// TwinCAT 3 PLC project PLC
// ProgramVersion: 3.1.4023.0
// libraries:
//   Tc2_Standard, * (Beckhoff Automation GmbH)
//   Tc2_System, * (Beckhoff Automation GmbH)
//   Tc3_Module, * (Beckhoff Automation GmbH)
// project tree:
//   / PlcTask.TcTTO
//   POUs/ MAIN.TcPOU
//   DUTs/IO/PdoEntries/ Status_56B69FDC.TcDUT (not stored), Inputs_62625F94.TcDUT (not stored), Ctrl_F19EAB21.TcDUT (not stored), Inputs_102D1D08.TcDUT (not stored), Status_642C2ED1.TcDUT (not stored), Ctrl_B05F80DF.TcDUT (not stored), Outputs_A910484D.TcDUT (not stored), Ctrl_77460BD3.TcDUT (not stored), Channel_EA8D33D7.TcDUT (not stored), Channel_D623F56C.TcDUT (not stored), Status_D9DC9C1B.TcDUT (not stored), Control_4E83000D.TcDUT (not stored), Status_8D3FCD23.TcDUT (not stored), Control_87176C1F.TcDUT (not stored), Device_status_8568DBCA.TcDUT (not stored), Outputs_Group_78994C08.TcDUT (not stored), Outputs_Channel_78994C08.TcDUT (not stored), Status_F2CE6D91.TcDUT (not stored), STATUS_B0753356.TcDUT (not stored), Status_237FCB0F.TcDUT (not stored), Setting_24C04940.TcDUT (not stored), Ctrl_56BB2DF2.TcDUT (not stored), Status_51F0A924.TcDUT (not stored), Settings_24C04940.TcDUT (not stored), Control_18D542D9.TcDUT (not stored), Status_439F40C3.TcDUT (not stored), Status_B0753356.TcDUT (not stored), Status_68C33E99.TcDUT (not stored), Status_7BCDA921.TcDUT (not stored), Ctrl_B9DDD3FF.TcDUT (not stored), Status_ACC8459F.TcDUT (not stored), Status_536663CA.TcDUT (not stored), Status_C03E2495.TcDUT (not stored), Status_A9D94975.TcDUT (not stored), Control_D500AB79.TcDUT (not stored), Status_81FEA767.TcDUT (not stored), Status_36731094.TcDUT (not stored), Status_6D6CFE20.TcDUT (not stored), Control_6EF2C5D0.TcDUT (not stored), Status_D8D782C3.TcDUT (not stored), Status_E2E79E85.TcDUT (not stored), Status_2E3946CF.TcDUT (not stored), Counter_value_E1FCE22B.TcDUT (not stored), Control_BD9A418F.TcDUT (not stored), Status_396FCBA0.TcDUT (not stored), Status_AA25F79C.TcDUT (not stored), Control_D4F3D880.TcDUT (not stored), Status_770B5231.TcDUT (not stored), Control_A35B59FC.TcDUT (not stored), Status_3E6F3FF3.TcDUT (not stored), Status_3BE3BF26.TcDUT (not stored), Control_135F4E52.TcDUT (not stored), Status_56494C1D.TcDUT (not stored), Status_3D84275F.TcDUT (not stored), Ctrl_71604E86.TcDUT (not stored), Ctrl_1EFB4D3B.TcDUT (not stored), Status_E3E7FD12.TcDUT (not stored), Slave_1_Inputs_2C3058A8.TcDUT (not stored), Slave_2_Inputs_413F454C.TcDUT (not stored), Slave_3_Inputs_9985457D.TcDUT (not stored), Slave_4_Inputs_9B217E84.TcDUT (not stored), Slave_5_Inputs_439B7EB5.TcDUT (not stored), Slave_6_Inputs_2E946351.TcDUT (not stored), Slave_7_Inputs_F62E6360.TcDUT (not stored), Slave_8_Inputs_2BDC14A3.TcDUT (not stored), Slave_9_Inputs_F3661492.TcDUT (not stored), Slave_10_Inputs_01E65E7D.TcDUT (not stored), Slave_11_Inputs_D274DB97.TcDUT (not stored), Slave_12_Inputs_A202481E.TcDUT (not stored), Slave_13_Inputs_7190CDF4.TcDUT (not stored), Slave_14_Inputs_42EF6F0C.TcDUT (not stored), Slave_15_Inputs_917DEAE6.TcDUT (not stored), Slave_16_Inputs_E10B796F.TcDUT (not stored), Slave_17_Inputs_3299FC85.TcDUT (not stored), Slave_18_Inputs_87F43C9F.TcDUT (not stored), Slave_19_Inputs_5466B975.TcDUT (not stored), Slave_20_Inputs_97C1CA9A.TcDUT (not stored), Slave_21_Inputs_44534F70.TcDUT (not stored), Slave_22_Inputs_3425DCF9.TcDUT (not stored), Slave_23_Inputs_E7B75913.TcDUT (not stored), Slave_24_Inputs_D4C8FBEB.TcDUT (not stored), Slave_25_Inputs_075A7E01.TcDUT (not stored), Slave_26_Inputs_772CED88.TcDUT (not stored), Slave_27_Inputs_A4BE6862.TcDUT (not stored), Slave_28_Inputs_11D3A878.TcDUT (not stored), Slave_29_Inputs_C2412D92.TcDUT (not stored), Slave_30_Inputs_199C4DAA.TcDUT (not stored), Slave_31_Inputs_CA0EC840.TcDUT (not stored), Slave_1_Outputs_820A30FD.TcDUT (not stored), Slave_2_Outputs_EF052D19.TcDUT (not stored), Slave_3_Outputs_37BF2D28.TcDUT (not stored), Slave_4_Outputs_351B16D1.TcDUT (not stored), Slave_5_Outputs_EDA116E0.TcDUT (not stored), Slave_6_Outputs_80AE0B04.TcDUT (not stored), Slave_7_Outputs_58140B35.TcDUT (not stored), Slave_8_Outputs_85E67CF6.TcDUT (not stored), Slave_9_Outputs_5D5C7CC7.TcDUT (not stored), Slave_10_Outputs_0FEEBBCA.TcDUT (not stored), Slave_11_Outputs_DC7C3E20.TcDUT (not stored), Slave_12_Outputs_AC0AADA9.TcDUT (not stored), Slave_13_Outputs_7F982843.TcDUT (not stored), Slave_14_Outputs_4CE78ABB.TcDUT (not stored), Slave_15_Outputs_9F750F51.TcDUT (not stored), Slave_16_Outputs_EF039CD8.TcDUT (not stored), Slave_17_Outputs_3C911932.TcDUT (not stored), Slave_18_Outputs_89FCD928.TcDUT (not stored), Slave_19_Outputs_5A6E5CC2.TcDUT (not stored), Slave_20_Outputs_99C92F2D.TcDUT (not stored), Slave_21_Outputs_4A5BAAC7.TcDUT (not stored), Slave_22_Outputs_3A2D394E.TcDUT (not stored), Slave_23_Outputs_E9BFBCA4.TcDUT (not stored), Slave_24_Outputs_DAC01E5C.TcDUT (not stored), Slave_25_Outputs_09529BB6.TcDUT (not stored), Slave_26_Outputs_7924083F.TcDUT (not stored), Slave_27_Outputs_AAB68DD5.TcDUT (not stored), Slave_28_Outputs_1FDB4DCF.TcDUT (not stored), Slave_29_Outputs_CC49C825.TcDUT (not stored), Slave_30_Outputs_1794A81D.TcDUT (not stored), Slave_31_Outputs_C4062DF7.TcDUT (not stored), Status_182674C6.TcDUT (not stored), Status_B6795845.TcDUT (not stored), Control_F189B737.TcDUT (not stored), Control_C948E0F2.TcDUT (not stored), Status_8CBE219F.TcDUT (not stored), Status_1E008DB9.TcDUT (not stored), Control_5FD4673D.TcDUT (not stored), Status_36C8BFF1.TcDUT (not stored), Status_FCAFFB9E.TcDUT (not stored), Control_534FEB19.TcDUT (not stored), Status_1D9409A4.TcDUT (not stored), Status_26C2D68E.TcDUT (not stored), Control_854091F6.TcDUT (not stored), Status_8AD1B54B.TcDUT (not stored), Control_0B2F8B70.TcDUT (not stored), FSOE_8C3E79C6.TcDUT (not stored), FSOE_3054F843.TcDUT (not stored), Status_8A0522A0.TcDUT (not stored), Ctrl_8F963B2D.TcDUT (not stored), Status_FCC1AD92.TcDUT (not stored), Status_6F0FEDB3.TcDUT (not stored), Control_DAEE1D52.TcDUT (not stored), Status_5E172F14.TcDUT (not stored), Status_CDD96F35.TcDUT (not stored), Status_B8381171.TcDUT (not stored), Status_7097155E.TcDUT (not stored), Control_7786EF9F.TcDUT (not stored), Status_70E023F8.TcDUT (not stored), Control_A8DDCD82.TcDUT (not stored), Status_EBCAF3EC.TcDUT (not stored), Control_254441A5.TcDUT (not stored), Status_72C27E80.TcDUT (not stored), Status_6BD97C37.TcDUT (not stored), Status_3BF44A81.TcDUT (not stored), Control_7648F432.TcDUT (not stored), Status_9AF2E088.TcDUT (not stored), Control_12F99C76.TcDUT (not stored), FSOE_BDDA3532.TcDUT (not stored), FSOE_EE2DB9C3.TcDUT (not stored), FSOE_046F804E.TcDUT (not stored), FSOE_F7635245.TcDUT (not stored), Status_05CE4FB5.TcDUT (not stored), Ctrl_AEDC374E.TcDUT (not stored), STATUS_1538B4EA.TcDUT (not stored), STATUS_522E84CD.TcDUT (not stored), STATUS_58431BA9.TcDUT (not stored), Status_543010BE.TcDUT (not stored), Samples_F24E104A.TcDUT (not stored), StartTimeNextLatch_02E0C1C8.TcDUT (not stored), U1_STATUS_B0753356.TcDUT (not stored), U1_SAMPLES_2D13B74B.TcDUT (not stored), I1_STATUS_B0753356.TcDUT (not stored), I1_SAMPLES_2D13B74B.TcDUT (not stored), U2_STATUS_B0753356.TcDUT (not stored), U2_SAMPLES_2D13B74B.TcDUT (not stored), I2_STATUS_B0753356.TcDUT (not stored), I2_SAMPLES_2D13B74B.TcDUT (not stored), U3_STATUS_B0753356.TcDUT (not stored), U3_SAMPLES_2D13B74B.TcDUT (not stored), I3_STATUS_B0753356.TcDUT (not stored), I3_SAMPLES_2D13B74B.TcDUT (not stored), U1_Status_DC903920.TcDUT (not stored), U1_Samples_2D13B74B.TcDUT (not stored), I1_Status_DC903920.TcDUT (not stored), I1_Samples_2D13B74B.TcDUT (not stored), U2_Status_DC903920.TcDUT (not stored), U2_Samples_2D13B74B.TcDUT (not stored), I2_Status_DC903920.TcDUT (not stored), I2_Samples_2D13B74B.TcDUT (not stored), U3_Status_DC903920.TcDUT (not stored), U3_Samples_2D13B74B.TcDUT (not stored), I3_Status_DC903920.TcDUT (not stored), I3_Samples_2D13B74B.TcDUT (not stored), U1_Samples_25492287.TcDUT (not stored), I1_Samples_25492287.TcDUT (not stored), U2_Samples_25492287.TcDUT (not stored), I2_Samples_25492287.TcDUT (not stored), U3_Samples_25492287.TcDUT (not stored), I3_Samples_25492287.TcDUT (not stored), U1_Samples_1109DCAA.TcDUT (not stored), I1_Samples_1109DCAA.TcDUT (not stored), U2_Samples_1109DCAA.TcDUT (not stored), I2_Samples_1109DCAA.TcDUT (not stored), U3_Samples_1109DCAA.TcDUT (not stored), I3_Samples_1109DCAA.TcDUT (not stored), High_Current_Range_48967762.TcDUT (not stored), Status_7BCA2D07.TcDUT (not stored), Ctrl_E6581599.TcDUT (not stored), Status_3035BE2E.TcDUT (not stored), Control_4AE59EC2.TcDUT (not stored)
//   DUTs/IO/PDOs/ InfoData_6F19DB2B.TcDUT (not stored), Channel_830843C1.TcDUT (not stored), WcState_9091E0EB.TcDUT (not stored), Channel_31CEFA7F.TcDUT (not stored), EMPTY_STRUCTURE.TcDUT (not stored), DC_1A6E6625.TcDUT (not stored), InfoData_A7436BC6.TcDUT (not stored), Latch_8E413295.TcDUT (not stored), Latch_39BD7C7C.TcDUT (not stored), Latch_0465F916.TcDUT (not stored), Ch1_CycleCount_9DBE2BC5.TcDUT (not stored), Ch1_Input_FFC4CE24.TcDUT (not stored), Ch2_CycleCount_976A51B5.TcDUT (not stored), Ch2_Input_78ADA90C.TcDUT (not stored), NextSync1Time_EE185E17.TcDUT (not stored), MTI_Inputs_10x_Channel_C3ED30FD.TcDUT (not stored), MTI_Outputs_Channel_0F1028A1.TcDUT (not stored), InfoData_BEF6B88E.TcDUT (not stored), MTI_Inputs_1x_Channel_CC1B212F.TcDUT (not stored), MTO_Inputs_Channel_53C09E8B.TcDUT (not stored), MTO_Outputs_10x_Channel_232E0117.TcDUT (not stored), MTO_Outputs_10x_Channel_A3C0C022.TcDUT (not stored), Channel_42CA91F7.TcDUT (not stored), WcState_0B2B16F9.TcDUT (not stored), DIG_Diag_Inputs_58F3E2A8.TcDUT (not stored), DIG_Inputs_Device_A1F150A9.TcDUT (not stored), DIG_Outputs_F9744C66.TcDUT (not stored), InfoData_32EB74EA.TcDUT (not stored), Diag_A72B1E17.TcDUT (not stored), Channel_54BE63B3.TcDUT (not stored), DOX_Status_Channel_09DD45C8.TcDUT (not stored), DOX_Control_Channel_A74F2363.TcDUT (not stored), DOX_Status_Channel_6FDDBA98.TcDUT (not stored), DOX_Control_Channel_E6930641.TcDUT (not stored), DC_Sync_Activate_FA2D2910.TcDUT (not stored), DC_Sync_Start_9CCB0E51.TcDUT (not stored), DC_Sync_Start_E82E9233.TcDUT (not stored), Cycle_Counter_2C233804.TcDUT (not stored), Sample_3C4603C7.TcDUT (not stored), CycCount0_2C233804.TcDUT (not stored), Sample_0023574C.TcDUT (not stored), CycCount1_2C233804.TcDUT (not stored), Sample_07D5B44A.TcDUT (not stored), CycCount0_AF431CE0.TcDUT (not stored), CycCount1_A8B5FFE6.TcDUT (not stored), StartTimeNextOutput_228767F4.TcDUT (not stored), Inputs_298FB92D.TcDUT (not stored), DO_Inputs_Device_4A9049C5.TcDUT (not stored), DO_Group_1_Outputs_59D8C01C.TcDUT (not stored), DO_Group_2_Outputs_82808288.TcDUT (not stored), DIG_Diag_Inputs_F289D615.TcDUT (not stored), DIG_Outputs_B9300CB6.TcDUT (not stored), Diagnostic_A72B1E17.TcDUT (not stored), DO_Group_1_Outputs_07009A9C.TcDUT (not stored), DO_Group_2_Outputs_3033EF65.TcDUT (not stored), DO_Group_3_Outputs_22DD3C32.TcDUT (not stored), DO_Group_4_Outputs_5E550497.TcDUT (not stored), AI_Inputs_Channel_10B8F80A.TcDUT (not stored), AI_Inputs_Channel_45213104.TcDUT (not stored), AI_Inputs_45213104.TcDUT (not stored), Ch1_Status_75824485.TcDUT (not stored), Ch1_Sample_A71DD501.TcDUT (not stored), Ch2_Status_75824485.TcDUT (not stored), Ch2_Sample_9F6886E6.TcDUT (not stored), Next_Sync1_Time_434371C2.TcDUT (not stored), Sample_Count_C25D5F38.TcDUT (not stored), NextSync1Time_9AFDC275.TcDUT (not stored), Sample_Count_EA88CAD9.TcDUT (not stored), SAI_Inputs_3A838E11.TcDUT (not stored), SAI_Range_C3200E78.TcDUT (not stored), SAI_Range_3710D747.TcDUT (not stored), SAI_Inputs_84B29FE9.TcDUT (not stored), SAI_Range_BDBF6DA9.TcDUT (not stored), SAI_Range_2A187FC5.TcDUT (not stored), SAI_Feedback_BDBF6DA9.TcDUT (not stored), SAI_Inputs_Channel_9DCD6557.TcDUT (not stored), SAI_Range_Channel_BDBF6DA9.TcDUT (not stored), SAI_Inputs_Real_Channel_CCECF13D.TcDUT (not stored), AI_Standard_Channel_A8DF64E3.TcDUT (not stored), TC_Inputs_Channel_204FE750.TcDUT (not stored), AI_Standard_Channel_4A394481.TcDUT (not stored), RMB_Status_C0E100AA.TcDUT (not stored), RMB_Value_INT_E9189C4B.TcDUT (not stored), RMB_Control_CC49845C.TcDUT (not stored), AO_Output_Channel_BA7EBB7C.TcDUT (not stored), Channel_5F9B7EA6.TcDUT (not stored), Channel_4E63E14D.TcDUT (not stored), Channel_DD2C734A.TcDUT (not stored), SSI_Inputs_0E3D8E33.TcDUT (not stored), SSI_Inputs_3B70A311.TcDUT (not stored), SSI_Inputs_8BC18DAC.TcDUT (not stored), SSI_Inputs_Channel_0E3D8E33.TcDUT (not stored), SSI_Inputs_Channel_EDA16284.TcDUT (not stored), ENC_Status_1E2673DC.TcDUT (not stored), ENC_Control_64DD586E.TcDUT (not stored), FB_Inputs_Channel_74050988.TcDUT (not stored), IND_Inputs_Channel_BBE8401F.TcDUT (not stored), IND_Outputs_Channel_02FDE6C9.TcDUT (not stored), Channel_B90637B9.TcDUT (not stored), Channel_C6781B15.TcDUT (not stored), Inputs_B90637B9.TcDUT (not stored), Outputs_C6781B15.TcDUT (not stored), ENC_Status_compact_D1AA7539.TcDUT (not stored), ENC_Control_compact_6FDDC669.TcDUT (not stored), ENC_Status_compact_6F424558.TcDUT (not stored), ENC_Control_compact_21E2D14D.TcDUT (not stored), ENC_Status_compact_7D3464F3.TcDUT (not stored), ENC_Status_compact_4198EF3B.TcDUT (not stored), ENC_Status_4E2088B9.TcDUT (not stored), ENC_NextSync1Time_9AFDC275.TcDUT (not stored), ENC_TxPdo_1_Samples_Counter_value_215818C6.TcDUT (not stored), ENC_Control_14E3EF4F.TcDUT (not stored), ENC_Inputs_3399C5AA.TcDUT (not stored), ENC_Inputs_24B63C53.TcDUT (not stored), ENC_Outputs_2E45048F.TcDUT (not stored), ENC_Status_Channel_10A67E52.TcDUT (not stored), ENC_Control_Channel_4C8A7395.TcDUT (not stored), ENC_Status_Channel_04F16FC0.TcDUT (not stored), ENC_Control_Channel_B930862D.TcDUT (not stored), ENC_Inputs_561E041F.TcDUT (not stored), ENC_Inputs_B3536485.TcDUT (not stored), ENC_Outputs_21E2D14D.TcDUT (not stored), ENC_Status_AC51C0C0.TcDUT (not stored), ENC_Filtered_latch_2CF1EFF6.TcDUT (not stored), ENC_Control_EB665241.TcDUT (not stored), ENC_Inputs_F139456B.TcDUT (not stored), ENC_Outputs_6FDDC669.TcDUT (not stored), ENC_Status_compact_B3536485.TcDUT (not stored), ENC_Status_compact_Channel_0EF60376.TcDUT (not stored), ENC_Period_Channel_24B63C53.TcDUT (not stored), ENC_Control_compact_Channel_245CB94B.TcDUT (not stored), ENC_Status_compact_Channel_FA024B16.TcDUT (not stored), ENC_Control_compact_Channel_2ED727EF.TcDUT (not stored), Inputs_6C2FC202.TcDUT (not stored), Outputs_5D00B5E7.TcDUT (not stored), COM_Inputs_3801C95E.TcDUT (not stored), COM_Outputs_DEF408EC.TcDUT (not stored), COM_Inputs_Channel_3801C95E.TcDUT (not stored), COM_Outputs_Channel_EADA2E0D.TcDUT (not stored), COM_TxPDO_Map_Inputs_Channel_3801C95E.TcDUT (not stored), COM_RxPDO_Map_Outputs_Channel_EADA2E0D.TcDUT (not stored), COM_TxPDO_Map_Inputs_3801C95E.TcDUT (not stored), COM_RxPDO_Map_Outputs_DEF408EC.TcDUT (not stored), Status_EF5E6C28.TcDUT (not stored), Control_88301954.TcDUT (not stored), Status_07D3AAF6.TcDUT (not stored), Control_DAFD38E0.TcDUT (not stored), DIS_Inputs_E0E384E3.TcDUT (not stored), DIS_Outputs_6C9BFFEE.TcDUT (not stored), ASI_Inputs_Device_7F2828A5.TcDUT (not stored), ASI_Status_8C8FBBB4.TcDUT (not stored), ASI_Outputs_Device_16036E19.TcDUT (not stored), ASI_Control_F45BBE2B.TcDUT (not stored), ASI_Status_279C3903.TcDUT (not stored), ASI_Control_2BED1893.TcDUT (not stored), DeviceState_Inputs_4751FF76.TcDUT (not stored), InfoData_90184F0C.TcDUT (not stored), DeviceState_Inputs_Device_A1210598.TcDUT (not stored), Module_1_DeviceState_Inputs_Device_5322301C.TcDUT (not stored), Module_2_DeviceState_Inputs_BD6C7035.TcDUT (not stored), ENC_Status_compact_3C6E2C44.TcDUT (not stored), STM_Status_36ED096F.TcDUT (not stored), ENC_Control_compact_2E82BC43.TcDUT (not stored), STM_Control_5A8B5016.TcDUT (not stored), STM_Velocity_A47A3F41.TcDUT (not stored), InfoData_8DF4E0C5.TcDUT (not stored), InfoData_6538CF5F.TcDUT (not stored), AI_Standard_Channel_205D8A06.TcDUT (not stored), InfoData_939F71B6.TcDUT (not stored), ENC_Status_compact_4D066E1A.TcDUT (not stored), STM_Status_DE0D6B37.TcDUT (not stored), STM_Control_BA4CE352.TcDUT (not stored), STM_Status_5B5B2475.TcDUT (not stored), FB_Position_3FA094ED.TcDUT (not stored), DRV_Statusword_9B36FDFC.TcDUT (not stored), DRV_Following_error_actual_value_5AA320BF.TcDUT (not stored), DRV_Controlword_F3F14721.TcDUT (not stored), DRV_Target_position_05240F14.TcDUT (not stored), InfoData_6185D47C.TcDUT (not stored), PowerOK_830843C1.TcDUT (not stored), PowerOK_CEB2FD12.TcDUT (not stored), FuseError_1EC650DA.TcDUT (not stored), OCP_Inputs_8CCE65FB.TcDUT (not stored), OCP_Outputs_01014934.TcDUT (not stored), OCP_Inputs_Channel_8CCE65FB.TcDUT (not stored), OCP_Outputs_Channel_01014934.TcDUT (not stored), OCP_Inputs_Channel_794A321B.TcDUT (not stored), Status_Us_B1E819A2.TcDUT (not stored), Status_Up_B1E819A2.TcDUT (not stored), Status_Uo_B8D9F2FA.TcDUT (not stored), Status_Up_DB353128.TcDUT (not stored), Status_Us_DB353128.TcDUT (not stored), Status_Us_449D6AB5.TcDUT (not stored), Status_Uo_449D6AB5.TcDUT (not stored), BCT_Inputs_28C1780C.TcDUT (not stored), BCT_Inputs_8E55234D.TcDUT (not stored), BCT_Inputs_4B987895.TcDUT (not stored), BCT_Inputs_8B1D510C.TcDUT (not stored), BCT_Inputs_7ACE8FA6.TcDUT (not stored), CNT_Inputs_7D4495CD.TcDUT (not stored), CNT_Outputs_EB14A675.TcDUT (not stored), CNT_Inputs_147BF88E.TcDUT (not stored), CNT_Inputs_B6C38E71.TcDUT (not stored), CNT_Outputs_458039AE.TcDUT (not stored), CNT_Inputs_Channel_21E1BB39.TcDUT (not stored), CNT_Outputs_Channel_774A30BC.TcDUT (not stored), CNT_Inputs_Channel_54FF2F1E.TcDUT (not stored), CNT_Outputs_Channel_550BB6DF.TcDUT (not stored), FSoE_Inputs_8E27404E.TcDUT (not stored), FSoE_Outputs_5936ECC6.TcDUT (not stored), FSLOGIC_Inputs_EEE9388E.TcDUT (not stored), Module_1_FSOE_79A9B6A8.TcDUT (not stored), Module_2_FSLOGIC_DEAB4522.TcDUT (not stored), PWM_Outputs_Channel_4C6289CD.TcDUT (not stored), PWM_Inputs_Channel_4239F652.TcDUT (not stored), PWM_SysTime_Channel_10DC6945.TcDUT (not stored), PWM_Per_DC_Outputs_Channel_C8E719F3.TcDUT (not stored), Inputs_A3335424.TcDUT (not stored), Outputs_8F8B60FA.TcDUT (not stored), PTO_Status_B6D696E0.TcDUT (not stored), ENC_Status_compact_EA7A730E.TcDUT (not stored), PTO_Control_392B4D2E.TcDUT (not stored), PTO_Target_compact_5C359F7D.TcDUT (not stored), ENC_Control_compact_245CB94B.TcDUT (not stored), PTO_Status_B24E260C.TcDUT (not stored), ENC_Status_compact_4C428F88.TcDUT (not stored), PTO_Control_9287F8E4.TcDUT (not stored), ENC_Control_compact_2ED727EF.TcDUT (not stored), PTO_Status_40B3051C.TcDUT (not stored), ENC_Status_compact_036460C9.TcDUT (not stored), PTO_Status_C6D3EC31.TcDUT (not stored), ENC_Status_compact_64F890EB.TcDUT (not stored), PLS_Status_A60F4933.TcDUT (not stored), ENC_Control_compact_DC4E290B.TcDUT (not stored), PLS_Control_compact_DC91A7B8.TcDUT (not stored), PTO_Status_E0EB10E8.TcDUT (not stored), PLS_Status_70E7A1E2.TcDUT (not stored), PLS_Control_compact_CD6E44DE.TcDUT (not stored), Inputs_0292EF13.TcDUT (not stored), Outputs_905E7D86.TcDUT (not stored), PTO_Status_Channel_E0EB10E8.TcDUT (not stored), ENC_Status_Channel_A9252C48.TcDUT (not stored), PTO_Control_Channel_9287F8E4.TcDUT (not stored), PTO_Target_Channel_1F6D5BC6.TcDUT (not stored), ENC_Control_Channel_686BB9DC.TcDUT (not stored), PWM_Status_Channel_2D1AF340.TcDUT (not stored), PWM_Control_Channel_63F162E4.TcDUT (not stored), PWM_Status_Channel_77939B11.TcDUT (not stored), PWM_Inputs_Channel_304DC245.TcDUT (not stored), PWM_Outputs_Channel_D6F04FBD.TcDUT (not stored), DOX_Status_AED8A12A.TcDUT (not stored), DOX_Control_75D5C9E2.TcDUT (not stored), DOX_Status_F52B34D3.TcDUT (not stored), DOX_Control_B191BB93.TcDUT (not stored), FSoE_Inputs_C161D7C0.TcDUT (not stored), FSoE_Outputs_F73BE43A.TcDUT (not stored), Outputs_A2CAA446.TcDUT (not stored), FIELDVOLTAGE_Field_Voltage_Status_9DC7C349.TcDUT (not stored), WcState_B516A264.TcDUT (not stored), Module_1_FSOE_7E34DB40.TcDUT (not stored), Module_2_FSOUT_1E8D1637.TcDUT (not stored), Module_3_DEVICEIO_5FA6B4E7.TcDUT (not stored), Module_4_FSLOGIC_DEAB4522.TcDUT (not stored), FSoE_Inputs_939ABF3D.TcDUT (not stored), FSoE_Outputs_3899B185.TcDUT (not stored), Outputs_8B1C946D.TcDUT (not stored), Module_1_FSOE_263516AE.TcDUT (not stored), Module_2_FSOUT_6D5CB05D.TcDUT (not stored), AI_Standard_EA9DF21E.TcDUT (not stored), AI_Standard_Channel_EA9DF21E.TcDUT (not stored), AI_Standard_A8DF64E3.TcDUT (not stored), Channel_7539AA33.TcDUT (not stored), Ch_1_Al_Inputs_4794C083.TcDUT (not stored), Ch_2_Al_Inputs_4794C083.TcDUT (not stored), Ch_1_A1FAE759.TcDUT (not stored), Ch_2_D9CD36D2.TcDUT (not stored), RTD_Inputs_EA9DF21E.TcDUT (not stored), RTD_Inputs_Channel_EA9DF21E.TcDUT (not stored), RTD_Inputs_Channel_9575FEA1.TcDUT (not stored), RTD_Standard_Channel_A8DF64E3.TcDUT (not stored), AI_Compact_Channel_80E77D6A.TcDUT (not stored), TC_Inputs_EA9DF21E.TcDUT (not stored), TC_Inputs_Channel_EA9DF21E.TcDUT (not stored), TC_Inputs_Channel_45213104.TcDUT (not stored), TC_Channel_9575FEA1.TcDUT (not stored), AIBridge_Inputs_555AA1E8.TcDUT (not stored), AISupply_Inputs_555AA1E8.TcDUT (not stored), RMB_Control_4997AEF6.TcDUT (not stored), PM_Inputs_Channel_6909D406.TcDUT (not stored), PM_Status_data_0FD072A0.TcDUT (not stored), PM_Outputs_Channel_E5FBDE30.TcDUT (not stored), PM_Inputs_Channel_2468BF1D.TcDUT (not stored), PM_Inputs_Channel_2F868086.TcDUT (not stored), PM_Status_data_2A9514CB.TcDUT (not stored), PM_Inputs_Channel_345EAE54.TcDUT (not stored), PM_Inputs_Auxiliary_392D510B.TcDUT (not stored), PM_Outputs_Auxiliary_6BC1946F.TcDUT (not stored), PM_Inputs_Auxiliary_3661DB6D.TcDUT (not stored), Total_Status_1ACE98F0.TcDUT (not stored), Total_Advanced_3B87F467.TcDUT (not stored), Total_Active_C9A69AC1.TcDUT (not stored), Total_Apparent_8F93F985.TcDUT (not stored), Total_Reactive_EF01DEFD.TcDUT (not stored), Total_Statistic_Power_092925BE.TcDUT (not stored), Total_Statistic_PQF_E0243244.TcDUT (not stored), Total_Interval_Energy_37FCCEB0.TcDUT (not stored), Interval_1578BBD4.TcDUT (not stored), Total_Interval_1578BBD4.TcDUT (not stored), Total_Active_Reduced_0E616AE5.TcDUT (not stored), Total_Apparent_Reduced_4B7F3014.TcDUT (not stored), Total_Reactive_Reduced_207ED80C.TcDUT (not stored), Total_Interval_Energy_Reduced_B0A0CDD8.TcDUT (not stored), L1_Status_61BE8896.TcDUT (not stored), L1_Basic_665874DE.TcDUT (not stored), L1_Power_22301EDD.TcDUT (not stored), L1_Timing_CCFF711F.TcDUT (not stored), L2_Status_61BE8896.TcDUT (not stored), L2_Basic_665874DE.TcDUT (not stored), L2_Power_22301EDD.TcDUT (not stored), L2_Timing_CCFF711F.TcDUT (not stored), L3_Status_61BE8896.TcDUT (not stored), L3_Basic_665874DE.TcDUT (not stored), L3_Power_22301EDD.TcDUT (not stored), L3_Timing_CCFF711F.TcDUT (not stored), Total_Basic_FC2CFF17.TcDUT (not stored), Total_Active_F9B49EA1.TcDUT (not stored), Total_L_L_Voltage_28813519.TcDUT (not stored), Total_Total_L_L_Voltage_28813519.TcDUT (not stored), I1_Current_AFE1DFA2.TcDUT (not stored), I2_Current_AFE1DFA2.TcDUT (not stored), I3_Current_AFE1DFA2.TcDUT (not stored), I4_Current_AFE1DFA2.TcDUT (not stored), I5_Current_AFE1DFA2.TcDUT (not stored), I6_Current_AFE1DFA2.TcDUT (not stored), Total_Basic_F53F9C95.TcDUT (not stored), Total_Status_A62BD506.TcDUT (not stored), L1_Status_12B1E6BB.TcDUT (not stored), L2_Status_12B1E6BB.TcDUT (not stored), L3_Status_12B1E6BB.TcDUT (not stored), Total_Status_AD43C3B9.TcDUT (not stored), L1_Basic_9F3F6F48.TcDUT (not stored), L2_Basic_9F3F6F48.TcDUT (not stored), L3_Basic_9F3F6F48.TcDUT (not stored), PAI_Status_Channel_AE4AC104.TcDUT (not stored), PAI_Samples_EEA51725.TcDUT (not stored), PAI_Timestamp_6DC4D296.TcDUT (not stored), L1_Voltage_Status_784F03AD.TcDUT (not stored), L1_Voltage_Samples_ED678DEE.TcDUT (not stored), L1_Current_Samples_89E07818.TcDUT (not stored), L1_Current_Samples_3209B12F.TcDUT (not stored), L2_Voltage_Status_0626A010.TcDUT (not stored), L2_Voltage_Samples_D91109BE.TcDUT (not stored), L2_Current_Status_F789DBA5.TcDUT (not stored), L2_Current_Samples_067F357F.TcDUT (not stored), L3_Voltage_Status_2C01C17B.TcDUT (not stored), L3_Voltage_Samples_CAC3758E.TcDUT (not stored), L3_Current_Status_DDAEBACE.TcDUT (not stored), L3_Current_Samples_15AD494F.TcDUT (not stored), AI_Timestamp_NextSync1Time_9AFDC275.TcDUT (not stored), AI_CycleCount_B1A935A2.TcDUT (not stored), L1_Current_Status_89E07818.TcDUT (not stored), AI_Sample_Count_B1A935A2.TcDUT (not stored), L1_Voltage_Status_7371B043.TcDUT (not stored), L1_Voltage_Samples_926B408D.TcDUT (not stored), L1_Current_Status_82DECBF6.TcDUT (not stored), L1_Current_Samples_4D057C4C.TcDUT (not stored), L2_Voltage_Status_0D1813FE.TcDUT (not stored), L2_Voltage_Samples_A61DC4DD.TcDUT (not stored), L2_Current_Status_FCB7684B.TcDUT (not stored), L2_Current_Samples_7973F81C.TcDUT (not stored), L3_Voltage_Status_273F7295.TcDUT (not stored), L3_Voltage_Samples_B5CFB8ED.TcDUT (not stored), L3_Current_Status_D6900920.TcDUT (not stored), L3_Current_Samples_6AA1842C.TcDUT (not stored), AI_NextSync1Time_6DC4D296.TcDUT (not stored), AI_Sample_Count_EA88CAD9.TcDUT (not stored), L1_Voltage_Samples_41AEB7FF.TcDUT (not stored), L1_Current_Samples_9EC08B3E.TcDUT (not stored), L2_Voltage_Samples_75D833AF.TcDUT (not stored), L2_Current_Samples_AAB60F6E.TcDUT (not stored), L3_Voltage_Samples_660A4F9F.TcDUT (not stored), L3_Current_Samples_B964735E.TcDUT (not stored), L1_Voltage_Samples_A8076B5D.TcDUT (not stored), L1_Current_Samples_7769579C.TcDUT (not stored), L2_Voltage_Samples_9C71EF0D.TcDUT (not stored), L2_Current_Samples_431FD3CC.TcDUT (not stored), L3_Voltage_Samples_8FA3933D.TcDUT (not stored), L3_Current_Samples_50CDAFFC.TcDUT (not stored), AI_Current_Range_9DEBDE6D.TcDUT (not stored), Ch1_CycleCount_08F5A7EF.TcDUT (not stored), Ch1_Sample_C81C74F6.TcDUT (not stored), Ch2_CycleCount_0221DD9F.TcDUT (not stored), Ch2_Sample_F0692711.TcDUT (not stored), Sample_B442BB65.TcDUT (not stored), Status_D30DC33F.TcDUT (not stored), SYNC_Inputs_462ED321.TcDUT (not stored), SYNC_Inputs_1DE69B90.TcDUT (not stored), SYNC_Inputs_971453DD.TcDUT (not stored), External_Sync_69535D98.TcDUT (not stored), DMX_Status_5716F9AF.TcDUT (not stored), DMX_Control_8D35CC31.TcDUT (not stored), DMX_Channel_FF1F0CB6.TcDUT (not stored), DMX_Channel_DC7E3036.TcDUT (not stored), DMX_Channel_60D8A7A5.TcDUT (not stored), DMX_Channel_AEBD2226.TcDUT (not stored), DMX_Channel_346A633C.TcDUT (not stored), DMX_Channel_C9FE109C.TcDUT (not stored), DMX_Channel_A44FB6B6.TcDUT (not stored), DMX_Channel_BD63FDF6.TcDUT (not stored), DMX_Status_5ECDEABE.TcDUT (not stored), DMX_Channel_005FDEFD.TcDUT (not stored), COM_TxPDO_Map_Inputs_93BAD1D7.TcDUT (not stored), COM_RxPDO_Map_01DE24DC.TcDUT (not stored), DEVICE_Inputs_745C19EA.TcDUT (not stored), DEVICE_Outputs_DAFD38E0.TcDUT (not stored), DRV_Target_velocity_08A9583B.TcDUT (not stored), InfoData_96C94FAE.TcDUT (not stored), DS402_Statusword_9B36FDFC.TcDUT (not stored), DS402_Position_actual_value_07DC4C74.TcDUT (not stored), DS402_Controlword_F3F14721.TcDUT (not stored), DS402_Target_velocity_08A9583B.TcDUT (not stored), DCM_Status_Channel_36ED096F.TcDUT (not stored), DCM_Control_Channel_5A8B5016.TcDUT (not stored), DCM_Velocity_Channel_A47A3F41.TcDUT (not stored), ENC_Status_compact_Channel_DC559AB0.TcDUT (not stored), ENC_Control_compact_Channel_2E82BC43.TcDUT (not stored), DCM_Control_Channel_94BFDFDF.TcDUT (not stored), InfoData_E68C61CD.TcDUT (not stored), InfoData_2A97D6CF.TcDUT (not stored), Inputs_25A0042B.TcDUT (not stored), Outputs_2397A10E.TcDUT (not stored)
//   DUTs/IO/Boxes/ EK1100_1FC0878B.TcDUT, EK1122_1FC0878B.TcDUT, EL1002_02444DCB.TcDUT, EL1004_D135F8DB.TcDUT, EL1008_78E8D3DD.TcDUT, EL1012_02444DCB.TcDUT, EL1014_D135F8DB.TcDUT, EL1018_78E8D3DD.TcDUT, EL1024_D135F8DB.TcDUT, EL1034_D135F8DB.TcDUT, EL1052_6CC2DB6A.TcDUT, EL1054_37C87A1C.TcDUT, EL1084_D135F8DB.TcDUT, EL1088_78E8D3DD.TcDUT, EL1094_D135F8DB.TcDUT, EL1098_78E8D3DD.TcDUT, EL1104_D135F8DB.TcDUT, EL1114_D135F8DB.TcDUT, EL1124_D135F8DB.TcDUT, EL1134_D135F8DB.TcDUT, EL1144_D135F8DB.TcDUT, EL1202_02444DCB.TcDUT, EL1202_647E4607.TcDUT, EL1252_0C2D47B4.TcDUT, EL1252_934A18FC.TcDUT, EL1254_D5E6FA5F.TcDUT, EL1262_0FA571DE.TcDUT, EL1258_733F03F2.TcDUT, EL1258_699E7002.TcDUT, EL1259_5165368D.TcDUT, EL1259_AB1DE4FC.TcDUT, EL1382_6CC2DB6A.TcDUT, EL1702_02444DCB.TcDUT, EL1712_02444DCB.TcDUT, EL1722_02444DCB.TcDUT, EL1804_D135F8DB.TcDUT, EL1808_78E8D3DD.TcDUT, EL1809_32157CFD.TcDUT, EL1814_D135F8DB.TcDUT, EL1819_32157CFD.TcDUT, EL1852_7699BCF6.TcDUT, EL1859_7699BCF6.TcDUT, EL1862_32157CFD.TcDUT, EL1872_32157CFD.TcDUT, EL1889_32157CFD.TcDUT, EL1899_32157CFD.TcDUT, EL2002_B0214940.TcDUT, EL2004_7B64371E.TcDUT, EL2008_E2806B95.TcDUT, EL2014_12F3E4E3.TcDUT, EL2022_B0214940.TcDUT, EL2024_7B64371E.TcDUT, EL2032_4C3AB2A4.TcDUT, EL2034_9227BD07.TcDUT, EL2042_B0214940.TcDUT, EL2044_12F3E4E3.TcDUT, EL2084_7B64371E.TcDUT, EL2088_E2806B95.TcDUT, EL2124_7B64371E.TcDUT, EL2202_B0214940.TcDUT, EL2202_E4D0F256.TcDUT, EL2202_FB12F0C6.TcDUT, EL2212_25BC0E0A.TcDUT, EL2212_C6DE6766.TcDUT, EL2252_FF939DB0.TcDUT, EL2252_BD1134C6.TcDUT, EL2252_F49A8E92.TcDUT, EL2258_1A7A2033.TcDUT, EL2258_41B36B91.TcDUT, EL2262_4683CFC9.TcDUT, EL2262_79C970B1.TcDUT, EL2262_147DB6E1.TcDUT, EL2262_9619875D.TcDUT, EL2602_B0214940.TcDUT, EL2602_47E63F27.TcDUT, EL2612_B0214940.TcDUT, EL2622_B0214940.TcDUT, EL2622_47E63F27.TcDUT, EL2624_7B64371E.TcDUT, EL2634_7B64371E.TcDUT, EL2642_C5F9ACE7.TcDUT, EL2652_B0214940.TcDUT, EL2712_B0214940.TcDUT, EL2722_B0214940.TcDUT, EL2732_B0214940.TcDUT, EL2784_7B64371E.TcDUT, EL2788_E2806B95.TcDUT, EL2794_7B64371E.TcDUT, EL2798_E2806B95.TcDUT, EL2808_E2806B95.TcDUT, EL2809_2B6483BD.TcDUT, EL2819_3C4AB9A7.TcDUT, EL2828_E2806B95.TcDUT, EL2872_2B6483BD.TcDUT, EL2878_76DE585D.TcDUT, EL2889_2B6483BD.TcDUT, ELM2642_AD2D58FD.TcDUT (not stored), ELM2644_9E566A2A.TcDUT (not stored), ELM2742_AD2D58FD.TcDUT (not stored), ELM2744_9E566A2A.TcDUT (not stored), EL3602_248DA72D.TcDUT (not stored), EL3602_308B0EAB.TcDUT (not stored), EL3611_707BD392.TcDUT (not stored), EL3612_248DA72D.TcDUT (not stored), EL3621_707BD392.TcDUT (not stored), EL3632_AD8E17EA.TcDUT (not stored), EL3632_E2B98A5C.TcDUT (not stored), EL3681_02A14E64.TcDUT (not stored), EL3681_0095B62C.TcDUT (not stored), EL3681_C165473F.TcDUT (not stored), EL3692_E2582216.TcDUT (not stored), EL3174_DCC78662.TcDUT, EL3314_C9476E1C.TcDUT, EL3201_F37BFE85.TcDUT, EL3202_27F12237.TcDUT, EL3356_1EAAA6FF.TcDUT, EL4001_B44B6D4B.TcDUT (not stored), EL4002_11E38659.TcDUT (not stored), EL4002_5AE37D91.TcDUT (not stored), EL4004_AB92710E.TcDUT (not stored), EL4004_15C7AA14.TcDUT (not stored), EL4008_4E77D882.TcDUT (not stored), EL4008_B1FEBD99.TcDUT (not stored), EL4011_B44B6D4B.TcDUT (not stored), EL4012_11E38659.TcDUT (not stored), EL4012_5AE37D91.TcDUT (not stored), EL4014_AB92710E.TcDUT (not stored), EL4014_15C7AA14.TcDUT (not stored), EL4018_4E77D882.TcDUT (not stored), EL4018_B1FEBD99.TcDUT (not stored), EL4021_B44B6D4B.TcDUT (not stored), EL4022_11E38659.TcDUT (not stored), EL4022_5AE37D91.TcDUT (not stored), EL4024_AB92710E.TcDUT (not stored), EL4024_15C7AA14.TcDUT (not stored), EL4028_4E77D882.TcDUT (not stored), EL4028_B1FEBD99.TcDUT (not stored), EL4031_B44B6D4B.TcDUT (not stored), EL4032_11E38659.TcDUT (not stored), EL4032_5AE37D91.TcDUT (not stored), EL4034_AB92710E.TcDUT (not stored), EL4034_15C7AA14.TcDUT (not stored), EL4038_4E77D882.TcDUT (not stored), EL4038_B1FEBD99.TcDUT (not stored), EL4102_2970C32C.TcDUT (not stored), EL4104_15C7AA14.TcDUT (not stored), EL4112_2970C32C.TcDUT (not stored), EL4114_15C7AA14.TcDUT (not stored), EL4122_2970C32C.TcDUT (not stored), EL4124_15C7AA14.TcDUT (not stored), EL4132_2970C32C.TcDUT (not stored), EL4134_15C7AA14.TcDUT (not stored), EL5001_51F879D6.TcDUT (not stored), EL5001_B186A7F4.TcDUT (not stored), EL5001_0B28D087.TcDUT (not stored), EL5001_E6AEC0B9.TcDUT (not stored), EL5001_3E8227ED.TcDUT (not stored), EL5002_6DCBC4C0.TcDUT (not stored), EL5002_31A396E2.TcDUT (not stored), EL5021_23D26521.TcDUT (not stored), EL5032_6C2441B0.TcDUT (not stored), EL5042_6C2441B0.TcDUT (not stored), EL5072_1878E756.TcDUT (not stored), EL5101_127DF9F1.TcDUT (not stored), EL5101_227F83AA.TcDUT (not stored), EL5101_9D67C241.TcDUT (not stored), EL5101_671C8D14.TcDUT (not stored), EL5101_7476E948.TcDUT (not stored), EL5101_382A92AF.TcDUT (not stored), EL5101_94ED0CD9.TcDUT (not stored), EL5151_84FDBA5C.TcDUT (not stored), EL5102_7F96361B.TcDUT (not stored), EL5112_85F35646.TcDUT (not stored), EL5122_7F22C2A7.TcDUT (not stored), EL5151_93354628.TcDUT (not stored), EL5151_905C5FD8.TcDUT (not stored), EL5151_28650B83.TcDUT (not stored), EL5151_27CA2A4C.TcDUT (not stored), EL5151_4D0E77FC.TcDUT (not stored), EL5151_8822C7D7.TcDUT (not stored), EL5152_68AD847E.TcDUT (not stored), EL5152_735D68BF.TcDUT (not stored), EL6001_C5ADEF9E.TcDUT (not stored), EL6001_B592E1CA.TcDUT (not stored), EL6002_D5B468BD.TcDUT (not stored), EL6002_81703A53.TcDUT (not stored), EL6021_C5ADEF9E.TcDUT (not stored), EL6021_B592E1CA.TcDUT (not stored), EL6021_4CB9967B.TcDUT (not stored), EL6022_D5B468BD.TcDUT (not stored), EL6070_EEB2FEF4.TcDUT (not stored), EL6080_BB2AF530.TcDUT (not stored), EL6080_9D61BA3F.TcDUT (not stored), EL6090_18BD01E9.TcDUT (not stored), EL6201_12FC4F5D.TcDUT (not stored), EL6201_F71597F7.TcDUT (not stored), EL6224_DFFBB702.TcDUT (not stored), EL6224_EDFF9F2F.TcDUT (not stored), EL6224_98EF2419.TcDUT (not stored), EL7031_AAA74C59.TcDUT (not stored), EL7031_022B4804.TcDUT (not stored), EL7031_B94C4934.TcDUT (not stored), EL7037_3E4BEAEF.TcDUT (not stored), EL7041_6D538C60.TcDUT (not stored), EL7041_C5DF883D.TcDUT (not stored), EL7041_B394362F.TcDUT (not stored), EL7041_1B183272.TcDUT (not stored), EL7041_022B4804.TcDUT (not stored), EL7047_3E4BEAEF.TcDUT (not stored), EL7411_236AD61B.TcDUT (not stored), EL9110_2DA353FE.TcDUT (not stored), EL9160_2DA353FE.TcDUT (not stored), EL9210_B3C0CA83.TcDUT (not stored), EL9221_8223B8D7.TcDUT (not stored), EL9222_621C429E.TcDUT (not stored), EL9227_5EE3BA1D.TcDUT (not stored), EL9260_B3C0CA83.TcDUT (not stored), EL9410_6BC01D14.TcDUT (not stored), EL9505_19A4723D.TcDUT (not stored), EL9508_19A4723D.TcDUT (not stored), EL9510_19A4723D.TcDUT (not stored), EL9512_19A4723D.TcDUT (not stored), EL9515_19A4723D.TcDUT (not stored), EL9520_C0C35FE8.TcDUT (not stored), EL9540_67D07E0A.TcDUT (not stored), EL9550_3E8321A9.TcDUT (not stored), EL9560_DD45A30A.TcDUT (not stored), EL9576_1C514380.TcDUT (not stored), EL9576_6D7359CA.TcDUT (not stored), EL9576_85AB5804.TcDUT (not stored), EL9576_1017F4A5.TcDUT (not stored), EL9576_C42142C6.TcDUT (not stored), EL9070_374A9F23.TcDUT (not stored), EL9080_8ACDA20B.TcDUT (not stored), EL9100_015D4DDE.TcDUT (not stored), EL9150_9660ADAB.TcDUT (not stored), EL9250_94095822.TcDUT (not stored), EL9180_8B150E8C.TcDUT (not stored), EL9181_8FD4133B.TcDUT (not stored), EL9182_829735E2.TcDUT (not stored), EL9183_86562855.TcDUT (not stored), EL9184_98117850.TcDUT (not stored), EL9185_9CD065E7.TcDUT (not stored), EL9186_9193433E.TcDUT (not stored), EL9187_95525E89.TcDUT (not stored), EL9188_AD1DE334.TcDUT (not stored), EL9189_A9DCFE83.TcDUT (not stored), EL9190_590CCF50.TcDUT (not stored), EL9195_4EC9A43B.TcDUT (not stored), EL9200_0334B857.TcDUT (not stored), EL9290_5B653AD9.TcDUT (not stored), EL9400_07E75345.TcDUT (not stored), EL9540_431BDE6B.TcDUT (not stored), EL9550_91021FB7.TcDUT (not stored), EL9570_31F081B8.TcDUT (not stored), EL9010_D29C2085.TcDUT (not stored), EL1502_55AAB421.TcDUT, EL1502_0B55A582.TcDUT, EL1502_160D2F0C.TcDUT, EL1512_FBA8C099.TcDUT, EL1512_47F42F75.TcDUT, EL1918_414C8426.TcDUT, EL2502_FE2154F7.TcDUT, EL2502_CC10C1AB.TcDUT, EL2521_68CF8E5F.TcDUT, EL2521_0D912D3B.TcDUT, EL2521_BB8FCF63.TcDUT, EL2521_07DB1BED.TcDUT, EL2521_E1428158.TcDUT, EL2521_2E43D334.TcDUT, EL2521_552DEED5.TcDUT, EL2522_EF4C90EB.TcDUT, EL2535_4F3A6797.TcDUT, EL2535_A64DD997.TcDUT, EL2564_18497D6E.TcDUT, EL2595_D1BA4B80.TcDUT, EL2595_54F09154.TcDUT, EL2596_0DFAD775.TcDUT, EL2911_3424714D.TcDUT, EL2912_BFF8CF19.TcDUT, EL3001_6939453A.TcDUT, EL3001_E22DFA28.TcDUT, EL3002_FF9B4B04.TcDUT, EL3002_63BCF660.TcDUT, EL3004_E8149C1F.TcDUT, EL3004_C4269E32.TcDUT, EL3008_E17B118E.TcDUT, EL3008_335F857B.TcDUT, EL3011_E22DFA28.TcDUT, EL3012_63BCF660.TcDUT, EL3014_C4269E32.TcDUT, EL3021_E22DFA28.TcDUT, EL3022_63BCF660.TcDUT, EL3024_C4269E32.TcDUT, EL3041_6939453A.TcDUT, EL3041_E22DFA28.TcDUT, EL3042_FF9B4B04.TcDUT, EL3042_63BCF660.TcDUT, EL3044_E8149C1F.TcDUT, EL3044_C4269E32.TcDUT, EL3048_E17B118E.TcDUT, EL3048_335F857B.TcDUT, EL3051_6939453A.TcDUT, EL3051_E22DFA28.TcDUT, EL3052_FF9B4B04.TcDUT, EL3052_63BCF660.TcDUT, EL3054_E8149C1F.TcDUT, EL3054_C4269E32.TcDUT, EL3058_E17B118E.TcDUT, EL3058_335F857B.TcDUT, EL3061_6939453A.TcDUT, EL3061_E22DFA28.TcDUT, EL3062_FF9B4B04.TcDUT, EL3062_63BCF660.TcDUT, EL3064_E8149C1F.TcDUT, EL3064_C4269E32.TcDUT, EL3068_E17B118E.TcDUT, EL3068_335F857B.TcDUT, EL3101_ADDA2D08.TcDUT, EL3102_80DA0D1B.TcDUT, EL3102_AA20D87B.TcDUT, EL3104_DCC78662.TcDUT, EL3111_ADDA2D08.TcDUT, EL3112_80DA0D1B.TcDUT, EL3112_AA20D87B.TcDUT, EL3114_DCC78662.TcDUT, EL3121_ADDA2D08.TcDUT, EL3122_80DA0D1B.TcDUT, EL3122_AA20D87B.TcDUT, EL3124_DCC78662.TcDUT, EL3141_ADDA2D08.TcDUT, EL3142_80DA0D1B.TcDUT, EL3142_AA20D87B.TcDUT, EL3144_DCC78662.TcDUT, EL3151_ADDA2D08.TcDUT, EL3152_80DA0D1B.TcDUT, EL3152_AA20D87B.TcDUT, EL3154_DCC78662.TcDUT, EL3161_ADDA2D08.TcDUT, EL3162_80DA0D1B.TcDUT, EL3162_AA20D87B.TcDUT, EL3164_DCC78662.TcDUT, EL3182_EF3C9D49.TcDUT, EL3201_771154E1.TcDUT, EL3202_75835C5C.TcDUT, EL3204_6F0438BE.TcDUT, EL3204_B6248F5B.TcDUT, EL3204_988CC224.TcDUT, EL3204_8BBE23EA.TcDUT, EL3208_E885804F.TcDUT, EL3214_8BBE23EA.TcDUT, EL3218_E885804F.TcDUT, EL3255_70670831.TcDUT, EL3255_1972F7C0.TcDUT, EL3255_B4D4BD51.TcDUT, EL3311_768B3E67.TcDUT, EL3311_18A81F50.TcDUT, EL3312_48655483.TcDUT, EL3312_BE98AB26.TcDUT, EL3314_18BBAF47.TcDUT, EL3314_E65CDB1C.TcDUT, EL3314_6E4DFFE5.TcDUT, EL3318_44C149FC.TcDUT, EL3351_6847F283.TcDUT, EL3356_8E3EBEA0.TcDUT, EL3403_A37C91B8.TcDUT, EL3403_B537021B.TcDUT, EL3403_200C4240.TcDUT, EL3413_0563D894.TcDUT, EL3413_0EB67A0F.TcDUT, EL3423_D53556D0.TcDUT (not stored), EL3423_E7B0A427.TcDUT (not stored), EL3423_8ADF1317.TcDUT (not stored), EL3433_0EB67A0F.TcDUT (not stored), EL3443_696F77D6.TcDUT (not stored), EL3443_721200EE.TcDUT (not stored), EL3446_D94D3CBC.TcDUT (not stored), EL3453_C83104B4.TcDUT (not stored), EL3453_24373016.TcDUT (not stored), EL3483_E64A5C78.TcDUT (not stored), EL3483_2E666A7F.TcDUT (not stored), EL3483_A24D6565.TcDUT (not stored), EL3702_C321C591.TcDUT (not stored), EL3742_30F92DF7.TcDUT (not stored), EL3742_C321C591.TcDUT (not stored), EL3751_8C60EAE5.TcDUT (not stored), EL3773_D0D76902.TcDUT (not stored), EL3773_39B64C97.TcDUT (not stored), EL3773_6B2F401D.TcDUT (not stored), EL3773_5329C7E9.TcDUT (not stored), EL3783_5437254B.TcDUT (not stored), EL4712_4B3D3BDA.TcDUT (not stored), EL4732_6D12A07D.TcDUT (not stored), EL4732_4B3D3BDA.TcDUT (not stored), EL6690_3564888A.TcDUT (not stored), EL6692_F12D40B3.TcDUT (not stored), EL6695_258CDFB4.TcDUT (not stored), EL6601_EEB2FEF4.TcDUT (not stored), EL6614_EEB2FEF4.TcDUT (not stored), EL6631_210A1A8D.TcDUT (not stored), EL6652_210A1A8D.TcDUT (not stored), EL6688_8DEED677.TcDUT (not stored), EL6688_747A9CEE.TcDUT (not stored), EL6690_FD149FC2.TcDUT (not stored), EL6720_210A1A8D.TcDUT (not stored), EL6731_210A1A8D.TcDUT (not stored), EL6740_BB2AF530.TcDUT (not stored), EL6751_210A1A8D.TcDUT (not stored), EL6752_210A1A8D.TcDUT (not stored), EL6784_9D61BA3F.TcDUT (not stored), EL6851_936A5E5B.TcDUT (not stored), EL6851_29AB8840.TcDUT (not stored), EL6861_D2EC03B8.TcDUT (not stored), EL6900_0B6D4005.TcDUT (not stored), EL6910_CD4DE200.TcDUT (not stored), EL6930_0B6D4005.TcDUT (not stored), EL7201_CE650BCF.TcDUT (not stored), EL7201_7BF21317.TcDUT (not stored), EL7201_FC4732E8.TcDUT (not stored), EL7211_CE650BCF.TcDUT (not stored), EL7211_7BF21317.TcDUT (not stored), EL7211_FC4732E8.TcDUT (not stored), EL7221_CE650BCF.TcDUT (not stored), EL7221_7BF21317.TcDUT (not stored), EL7221_FC4732E8.TcDUT (not stored), EL7332_615C2CE5.TcDUT (not stored), EL7342_2AE9C6B3.TcDUT (not stored), EL7342_ADEFCF40.TcDUT (not stored), EL9930_77AEBA45.TcDUT (not stored), EL9930_07FC3A1D.TcDUT (not stored), EL9930_B8165E3C.TcDUT (not stored)
//   DUTs/IO/Devices/ SyncUnitTask_2D604ED5.TcDUT (not stored), SyncUnitTasks_6FEB8257.TcDUT (not stored), SyncUnits_9F8710E1.TcDUT (not stored)
//   DUTs/IO/Topology/ Beckhoff_EL1xxxEK1122_4D1603AD.TcDUT (not stored), Beckhoff_EL1xxx_3E37AACA.TcDUT (not stored), Beckhoff_EL2xxxEK1122_964E4139.TcDUT (not stored), Beckhoff_EL2xxx_F4C539CA.TcDUT (not stored), Beckhoff_EL3xxxEK1122_DF7980B5.TcDUT (not stored), Beckhoff_EL3xxx_05984D3D.TcDUT (not stored), Beckhoff_EL3xxx_0030EK1122_55DAE3CA.TcDUT (not stored), Beckhoff_EL3xxx_0030_C37B7D48.TcDUT (not stored), Beckhoff_EL4xxxEK1122_243FD9A6.TcDUT (not stored), Beckhoff_EL4xxx_44DCAF8D.TcDUT (not stored), Beckhoff_EL5xxxEK1122_6D08182A.TcDUT (not stored), Beckhoff_EL5xxx_A510F272.TcDUT (not stored), Beckhoff_EL6xxxEK1122_B6505ABE.TcDUT (not stored), Beckhoff_EL6xxx_5832F4A8.TcDUT (not stored), Beckhoff_EL7xxxEK1122_FF679B32.TcDUT (not stored), Beckhoff_EL7xxx_96878FD5.TcDUT (not stored), Beckhoff_EL9xxxEK1122_0D2A34A3.TcDUT (not stored), Beckhoff_EL9xxx_6E572B5F.TcDUT (not stored), Beckhoff_EL15xxEK1122_586CA173.TcDUT (not stored), Beckhoff_EL15xx_7FFDF3B3.TcDUT (not stored), Beckhoff_EL19xxEK1122_2AE5B579.TcDUT (not stored), Beckhoff_EL19xx_C9550BF7.TcDUT (not stored), Beckhoff_EL25xxEK1122_8334E3E7.TcDUT (not stored), Beckhoff_EL25xx_A1E3F918.TcDUT (not stored), Beckhoff_EL29xxEK1122_F1BDF7ED.TcDUT (not stored), Beckhoff_EL29xx_FCC67B44.TcDUT (not stored), Beckhoff_EL30xxEK1122_6D8563B7.TcDUT (not stored), Beckhoff_EL30xx_59D86529.TcDUT (not stored), Beckhoff_EL31xxEK1122_183B2500.TcDUT (not stored), Beckhoff_EL31xx_098DC56E.TcDUT (not stored), Beckhoff_EL32xxEK1122_86F9EED9.TcDUT (not stored), Beckhoff_EL32xx_A91E9D41.TcDUT (not stored), Beckhoff_EL33xxEK1122_F347A86E.TcDUT (not stored), Beckhoff_EL33xx_149C8FF5.TcDUT (not stored), Beckhoff_EL34xxEK1122_BFBD64DC.TcDUT (not stored), Beckhoff_EL34xx_5C8507D7.TcDUT (not stored), Beckhoff_EL37xxEK1122_217FAF05.TcDUT (not stored), Beckhoff_EL37xx_82AB11DA.TcDUT (not stored), Beckhoff_EL47xxEK1122_DA39F616.TcDUT (not stored), Beckhoff_EL47xx_F9F61196.TcDUT (not stored), Beckhoff_EL66xxEK1122_DCCAD5BD.TcDUT (not stored), Beckhoff_EL66xx_32F43B79.TcDUT (not stored), Beckhoff_EL67xxEK1122_4856750E.TcDUT (not stored), Beckhoff_EL67xx_9D033AAA.TcDUT (not stored), Beckhoff_EL68xxEK1122_A41DAADD.TcDUT (not stored), Beckhoff_EL68xx_6F206275.TcDUT (not stored), Beckhoff_EL69xxEK1122_D1A3EC6A.TcDUT (not stored), Beckhoff_EL69xx_55DE5C9C.TcDUT (not stored), Beckhoff_EL72xxEK1122_A6E7F55E.TcDUT (not stored), Beckhoff_EL72xx_566ED46D.TcDUT (not stored), Beckhoff_EL73xxEK1122_D359B3E9.TcDUT (not stored), Beckhoff_EL73xx_3D4E24E0.TcDUT (not stored), Beckhoff_EL99xxEK1122_6AD98277.TcDUT (not stored), A_0003_EL9930_0000_0017_96B57C1D.TcDUT (not stored), A_0001_EL9930_0000_0016_F7CB469B.TcDUT (not stored), Beckhoff_EL99xx_FA66A12D.TcDUT (not stored), EtherCAT_Master_ELxxxx_D0BA48C6.TcDUT (not stored)
//   DUTs/IO/Base/ EtcSlaveBase_82538BE2.TcDUT, EtcSlaveBase_82538BE2.TcDUT, EtcSlaveBase_82538BE2.TcDUT, EtcSlaveTerminalBase_947E5A46.TcDUT, EtcSlaveBoxBase_77A0E4A7.TcDUT, EtcSlaveEndTerminalBase_866C7F0C.TcDUT, InputBase_8311D824.TcDUT, OutputBase_10CEE7DE.TcDUT, EtcMasterBase_62654B43.TcDUT
//   GVLs/ GVL_iXlinker.TcGVL

CONFIGURATION PLC
    RESOURCE PLC ON TwinCAT3
        TASK PlcTask(INTERVAL := T#10ms, PRIORITY := 20);
        PROGRAM MAIN WITH PlcTask : MAIN;
    END_RESOURCE
END_CONFIGURATION

// ---- DUTs/IO/Boxes/EK1100_1FC0878B.TcDUT
{attribute 'GeneratedUsingTerminal: EK1100-0000-0018'}
{attribute addProperty BoxType "EK1100-0000-0018"}
{attribute addProperty Description "EK1100 EtherCAT Coupler (2A E-Bus)"}
{attribute addProperty Physics "YKY"}
{attribute addProperty Id "InfoDataAT %I*InfoData_6F19DB2B2"}
{attribute addProperty CRC "532711307"}
{attribute addProperty Size "2"}
TYPE EK1100_1FC0878B EXTENDS EtcSlaveBoxBase_77A0E4A7 :
STRUCT
	{attribute addProperty Name "InfoData"}
	InfoData : InfoData_6F19DB2B;
END_STRUCT
END_TYPE

// ---- DUTs/IO/Boxes/EK1122_1FC0878B.TcDUT
{attribute 'GeneratedUsingTerminal: EK1122-0000-0018'}
{attribute addProperty BoxType "EK1122-0000-0018"}
{attribute addProperty Description "EK1122 2 port EtherCAT junction"}
{attribute addProperty Physics "KYKY"}
{attribute addProperty Id "InfoDataAT %I*InfoData_6F19DB2B2"}
{attribute addProperty CRC "532711307"}
{attribute addProperty Size "2"}
TYPE EK1122_1FC0878B EXTENDS EtcSlaveTerminalBase_947E5A46 :
STRUCT
	{attribute addProperty Name "InfoData"}
	InfoData : InfoData_6F19DB2B;
END_STRUCT
END_TYPE

// ---- DUTs/IO/Boxes/EL1002_02444DCB.TcDUT
{attribute 'GeneratedUsingTerminal: EL1002--0000'}
{attribute addProperty BoxType "EL1002--0000"}
{attribute addProperty Description "EL1002 2Ch. Dig. Input 24V, 3ms"}
{attribute addProperty Physics "KK"}
{attribute addProperty Id "Channel_1AT %I*Channel_830843C11Channel_2AT %I*Channel_830843C11WcStateAT %I*WcState_9091E0EB2InfoDataAT %I*InfoData_6F19DB2B2"}
{attribute addProperty CRC "38030795"}
{attribute addProperty Size "6"}
TYPE EL1002_02444DCB EXTENDS EtcSlaveTerminalBase_947E5A46 :
STRUCT
	{attribute addProperty Name "Channel_1"}
	Channel_1 : Channel_830843C1;
	{attribute addProperty Name "Channel_2"}
	Channel_2 : Channel_830843C1;
	{attribute addProperty Name "WcState"}
	WcState : WcState_9091E0EB;
	{attribute addProperty Name "InfoData"}
	InfoData : InfoData_6F19DB2B;
END_STRUCT
END_TYPE

// ---- DUTs/IO/Boxes/EL1004_D135F8DB.TcDUT
{attribute 'GeneratedUsingTerminal: EL1004--0000'}
{attribute addProperty BoxType "EL1004--0000"}
{attribute addProperty Description "EL1004 4Ch. Dig. Input 24V, 3ms"}
{attribute addProperty Physics "KK"}
{attribute addProperty Id "Channel_1AT %I*Channel_830843C11Channel_2AT %I*Channel_830843C11Channel_3AT %I*Channel_830843C11Channel_4AT %I*Channel_830843C11WcStateAT %I*WcState_9091E0EB2InfoDataAT %I*InfoData_6F19DB2B2"}
{attribute addProperty CRC "3509975259"}
{attribute addProperty Size "8"}
TYPE EL1004_D135F8DB EXTENDS EtcSlaveTerminalBase_947E5A46 :
STRUCT
	{attribute addProperty Name "Channel_1"}
	Channel_1 : Channel_830843C1;
	{attribute addProperty Name "Channel_2"}
	Channel_2 : Channel_830843C1;
	{attribute addProperty Name "Channel_3"}
	Channel_3 : Channel_830843C1;
	{attribute addProperty Name "Channel_4"}
	Channel_4 : Channel_830843C1;
	{attribute addProperty Name "WcState"}
	WcState : WcState_9091E0EB;
	{attribute addProperty Name "InfoData"}
	InfoData : InfoData_6F19DB2B;
END_STRUCT
END_TYPE

// ---- DUTs/IO/Boxes/EL1008_78E8D3DD.TcDUT
{attribute 'GeneratedUsingTerminal: EL1008-0000-0016'}
{attribute addProperty BoxType "EL1008-0000-0016"}
{attribute addProperty Description "EL1008 8Ch. Dig. Input 24V, 3ms"}
{attribute addProperty Physics "KK"}
{attribute addProperty Id "Channel_1AT %I*Channel_830843C11Channel_2AT %I*Channel_830843C11Channel_3AT %I*Channel_830843C11Channel_4AT %I*Channel_830843C11Channel_5AT %I*Channel_830843C11Channel_6AT %I*Channel_830843C11Channel_7AT %I*Channel_830843C11Channel_8AT %I*Channel_830843C11WcStateAT %I*WcState_9091E0EB2InfoDataAT %I*InfoData_6F19DB2B2"}
{attribute addProperty CRC "2028524509"}
{attribute addProperty Size "12"}
TYPE EL1008_78E8D3DD EXTENDS EtcSlaveTerminalBase_947E5A46 :
STRUCT
	{attribute addProperty Name "Channel_1"}
	Channel_1 : Channel_830843C1;
	{attribute addProperty Name "Channel_2"}
	Channel_2 : Channel_830843C1;
	{attribute addProperty Name "Channel_3"}
	Channel_3 : Channel_830843C1;
	{attribute addProperty Name "Channel_4"}
	Channel_4 : Channel_830843C1;
	{attribute addProperty Name "Channel_5"}
	Channel_5 : Channel_830843C1;
	{attribute addProperty Name "Channel_6"}
	Channel_6 : Channel_830843C1;
	{attribute addProperty Name "Channel_7"}
	Channel_7 : Channel_830843C1;
	{attribute addProperty Name "Channel_8"}
	Channel_8 : Channel_830843C1;
	{attribute addProperty Name "WcState"}
	WcState : WcState_9091E0EB;
	{attribute addProperty Name "InfoData"}
	InfoData : InfoData_6F19DB2B;
END_STRUCT
END_TYPE

// ---- DUTs/IO/Boxes/EL1012_02444DCB.TcDUT
{attribute 'GeneratedUsingTerminal: EL1012--0000'}
{attribute addProperty BoxType "EL1012--0000"}
{attribute addProperty Description "EL1012 2Ch. Dig. Input 24V, 10µs"}
{attribute addProperty Physics "KK"}
{attribute addProperty Id "Channel_1AT %I*Channel_830843C11Channel_2AT %I*Channel_830843C11WcStateAT %I*WcState_9091E0EB2InfoDataAT %I*InfoData_6F19DB2B2"}
{attribute addProperty CRC "38030795"}
{attribute addProperty Size "6"}
TYPE EL1012_02444DCB EXTENDS EtcSlaveTerminalBase_947E5A46 :
STRUCT
	{attribute addProperty Name "Channel_1"}
	Channel_1 : Channel_830843C1;
	{attribute addProperty Name "Channel_2"}
	Channel_2 : Channel_830843C1;
	{attribute addProperty Name "WcState"}
	WcState : WcState_9091E0EB;
	{attribute addProperty Name "InfoData"}
	InfoData : InfoData_6F19DB2B;
END_STRUCT
END_TYPE

// ---- DUTs/IO/Boxes/EL1014_D135F8DB.TcDUT
{attribute 'GeneratedUsingTerminal: EL1014--0000'}
{attribute addProperty BoxType "EL1014--0000"}
{attribute addProperty Description "EL1014 4Ch. Dig. Input 24V, 10µs"}
{attribute addProperty Physics "KK"}
{attribute addProperty Id "Channel_1AT %I*Channel_830843C11Channel_2AT %I*Channel_830843C11Channel_3AT %I*Channel_830843C11Channel_4AT %I*Channel_830843C11WcStateAT %I*WcState_9091E0EB2InfoDataAT %I*InfoData_6F19DB2B2"}
{attribute addProperty CRC "3509975259"}
{attribute addProperty Size "8"}
TYPE EL1014_D135F8DB EXTENDS EtcSlaveTerminalBase_947E5A46 :
STRUCT
	{attribute addProperty Name "Channel_1"}
	Channel_1 : Channel_830843C1;
	{attribute addProperty Name "Channel_2"}
	Channel_2 : Channel_830843C1;
	{attribute addProperty Name "Channel_3"}
	Channel_3 : Channel_830843C1;
	{attribute addProperty Name "Channel_4"}
	Channel_4 : Channel_830843C1;
	{attribute addProperty Name "WcState"}
	WcState : WcState_9091E0EB;
	{attribute addProperty Name "InfoData"}
	InfoData : InfoData_6F19DB2B;
END_STRUCT
END_TYPE

// ---- DUTs/IO/Boxes/EL1018_78E8D3DD.TcDUT
{attribute 'GeneratedUsingTerminal: EL1018-0000-0016'}
{attribute addProperty BoxType "EL1018-0000-0016"}
{attribute addProperty Description "EL1018 8Ch. Dig. Input 24V, 10µs"}
{attribute addProperty Physics "KK"}
{attribute addProperty Id "Channel_1AT %I*Channel_830843C11Channel_2AT %I*Channel_830843C11Channel_3AT %I*Channel_830843C11Channel_4AT %I*Channel_830843C11Channel_5AT %I*Channel_830843C11Channel_6AT %I*Channel_830843C11Channel_7AT %I*Channel_830843C11Channel_8AT %I*Channel_830843C11WcStateAT %I*WcState_9091E0EB2InfoDataAT %I*InfoData_6F19DB2B2"}
{attribute addProperty CRC "2028524509"}
{attribute addProperty Size "12"}
TYPE EL1018_78E8D3DD EXTENDS EtcSlaveTerminalBase_947E5A46 :
STRUCT
	{attribute addProperty Name "Channel_1"}
	Channel_1 : Channel_830843C1;
	{attribute addProperty Name "Channel_2"}
	Channel_2 : Channel_830843C1;
	{attribute addProperty Name "Channel_3"}
	Channel_3 : Channel_830843C1;
	{attribute addProperty Name "Channel_4"}
	Channel_4 : Channel_830843C1;
	{attribute addProperty Name "Channel_5"}
	Channel_5 : Channel_830843C1;
	{attribute addProperty Name "Channel_6"}
	Channel_6 : Channel_830843C1;
	{attribute addProperty Name "Channel_7"}
	Channel_7 : Channel_830843C1;
	{attribute addProperty Name "Channel_8"}
	Channel_8 : Channel_830843C1;
	{attribute addProperty Name "WcState"}
	WcState : WcState_9091E0EB;
	{attribute addProperty Name "InfoData"}
	InfoData : InfoData_6F19DB2B;
END_STRUCT
END_TYPE

// ---- DUTs/IO/Boxes/EL1024_D135F8DB.TcDUT
{attribute 'GeneratedUsingTerminal: EL1024-0000-0016'}
{attribute addProperty BoxType "EL1024-0000-0016"}
{attribute addProperty Description "EL1024 4Ch. Dig. Input 24V, Type 2, 3ms"}
{attribute addProperty Physics "KK"}
{attribute addProperty Id "Channel_1AT %I*Channel_830843C11Channel_2AT %I*Channel_830843C11Channel_3AT %I*Channel_830843C11Channel_4AT %I*Channel_830843C11WcStateAT %I*WcState_9091E0EB2InfoDataAT %I*InfoData_6F19DB2B2"}
{attribute addProperty CRC "3509975259"}
{attribute addProperty Size "8"}
TYPE EL1024_D135F8DB EXTENDS EtcSlaveTerminalBase_947E5A46 :
STRUCT
	{attribute addProperty Name "Channel_1"}
	Channel_1 : Channel_830843C1;
	{attribute addProperty Name "Channel_2"}
	Channel_2 : Channel_830843C1;
	{attribute addProperty Name "Channel_3"}
	Channel_3 : Channel_830843C1;
	{attribute addProperty Name "Channel_4"}
	Channel_4 : Channel_830843C1;
	{attribute addProperty Name "WcState"}
	WcState : WcState_9091E0EB;
	{attribute addProperty Name "InfoData"}
	InfoData : InfoData_6F19DB2B;
END_STRUCT
END_TYPE

// ---- DUTs/IO/Boxes/EL1034_D135F8DB.TcDUT
{attribute 'GeneratedUsingTerminal: EL1034-0000-0016'}
{attribute addProperty BoxType "EL1034-0000-0016"}
{attribute addProperty Description "EL1034 4Ch. Dig. Input 24V, potential-free, 10µs"}
{attribute addProperty Physics "KK"}
{attribute addProperty Id "Channel_1AT %I*Channel_830843C11Channel_2AT %I*Channel_830843C11Channel_3AT %I*Channel_830843C11Channel_4AT %I*Channel_830843C11WcStateAT %I*WcState_9091E0EB2InfoDataAT %I*InfoData_6F19DB2B2"}
{attribute addProperty CRC "3509975259"}
{attribute addProperty Size "8"}
TYPE EL1034_D135F8DB EXTENDS EtcSlaveTerminalBase_947E5A46 :
STRUCT
	{attribute addProperty Name "Channel_1"}
	Channel_1 : Channel_830843C1;
	{attribute addProperty Name "Channel_2"}
	Channel_2 : Channel_830843C1;
	{attribute addProperty Name "Channel_3"}
	Channel_3 : Channel_830843C1;
	{attribute addProperty Name "Channel_4"}
	Channel_4 : Channel_830843C1;
	{attribute addProperty Name "WcState"}
	WcState : WcState_9091E0EB;
	{attribute addProperty Name "InfoData"}
	InfoData : InfoData_6F19DB2B;
END_STRUCT
END_TYPE

// ---- DUTs/IO/Boxes/EL1052_6CC2DB6A.TcDUT
{attribute 'GeneratedUsingTerminal: EL1052-0000-0016'}
{attribute addProperty BoxType "EL1052-0000-0016"}
{attribute addProperty Description "EL1052 2Ch. Dig. Input, NAMUR sensors"}
{attribute addProperty Physics "KK"}
{attribute addProperty Id "Channel_1AT %I*Channel_31CEFA7F2Channel_2AT %I*Channel_31CEFA7F2WcStateAT %I*WcState_9091E0EB2InfoDataAT %I*InfoData_6F19DB2B2"}
{attribute addProperty CRC "1824709482"}
{attribute addProperty Size "8"}
TYPE EL1052_6CC2DB6A EXTENDS EtcSlaveTerminalBase_947E5A46 :
STRUCT
	{attribute addProperty Name "Channel_1"}
	Channel_1 : Channel_31CEFA7F;
	{attribute addProperty Name "Channel_2"}
	Channel_2 : Channel_31CEFA7F;
	{attribute addProperty Name "WcState"}
	WcState : WcState_9091E0EB;
	{attribute addProperty Name "InfoData"}
	InfoData : InfoData_6F19DB2B;
END_STRUCT
END_TYPE

// ---- DUTs/IO/Boxes/EL1054_37C87A1C.TcDUT
{attribute 'GeneratedUsingTerminal: EL1054-0000-0016'}
{attribute addProperty BoxType "EL1054-0000-0016"}
{attribute addProperty Description "EL1054 4Ch. Dig. Input, NAMUR sensors"}
{attribute addProperty Physics "KK"}
{attribute addProperty Id "Channel_1AT %I*Channel_31CEFA7F2Channel_2AT %I*Channel_31CEFA7F2Channel_3AT %I*Channel_31CEFA7F2Channel_4AT %I*Channel_31CEFA7F2WcStateAT %I*WcState_9091E0EB2InfoDataAT %I*InfoData_6F19DB2B2"}
{attribute addProperty CRC "935885340"}
{attribute addProperty Size "12"}
TYPE EL1054_37C87A1C EXTENDS EtcSlaveTerminalBase_947E5A46 :
STRUCT
	{attribute addProperty Name "Channel_1"}
	Channel_1 : Channel_31CEFA7F;
	{attribute addProperty Name "Channel_2"}
	Channel_2 : Channel_31CEFA7F;
	{attribute addProperty Name "Channel_3"}
	Channel_3 : Channel_31CEFA7F;
	{attribute addProperty Name "Channel_4"}
	Channel_4 : Channel_31CEFA7F;
	{attribute addProperty Name "WcState"}
	WcState : WcState_9091E0EB;
	{attribute addProperty Name "InfoData"}
	InfoData : InfoData_6F19DB2B;
END_STRUCT
END_TYPE

// ---- DUTs/IO/Boxes/EL1084_D135F8DB.TcDUT
{attribute 'GeneratedUsingTerminal: EL1084-0000-0016'}
{attribute addProperty BoxType "EL1084-0000-0016"}
{attribute addProperty Description "EL1084 4Ch. Dig. Input 24V, 3ms, negative"}
{attribute addProperty Physics "KK"}
{attribute addProperty Id "Channel_1AT %I*Channel_830843C11Channel_2AT %I*Channel_830843C11Channel_3AT %I*Channel_830843C11Channel_4AT %I*Channel_830843C11WcStateAT %I*WcState_9091E0EB2InfoDataAT %I*InfoData_6F19DB2B2"}
{attribute addProperty CRC "3509975259"}
{attribute addProperty Size "8"}
TYPE EL1084_D135F8DB EXTENDS EtcSlaveTerminalBase_947E5A46 :
STRUCT
	{attribute addProperty Name "Channel_1"}
	Channel_1 : Channel_830843C1;
	{attribute addProperty Name "Channel_2"}
	Channel_2 : Channel_830843C1;
	{attribute addProperty Name "Channel_3"}
	Channel_3 : Channel_830843C1;
	{attribute addProperty Name "Channel_4"}
	Channel_4 : Channel_830843C1;
	{attribute addProperty Name "WcState"}
	WcState : WcState_9091E0EB;
	{attribute addProperty Name "InfoData"}
	InfoData : InfoData_6F19DB2B;
END_STRUCT
END_TYPE

// ---- DUTs/IO/Boxes/EL1088_78E8D3DD.TcDUT
{attribute 'GeneratedUsingTerminal: EL1088-0000-0016'}
{attribute addProperty BoxType "EL1088-0000-0016"}
{attribute addProperty Description "EL1088 8Ch. Dig. Input 24V, 3ms, negative"}
{attribute addProperty Physics "KK"}
{attribute addProperty Id "Channel_1AT %I*Channel_830843C11Channel_2AT %I*Channel_830843C11Channel_3AT %I*Channel_830843C11Channel_4AT %I*Channel_830843C11Channel_5AT %I*Channel_830843C11Channel_6AT %I*Channel_830843C11Channel_7AT %I*Channel_830843C11Channel_8AT %I*Channel_830843C11WcStateAT %I*WcState_9091E0EB2InfoDataAT %I*InfoData_6F19DB2B2"}
{attribute addProperty CRC "2028524509"}
{attribute addProperty Size "12"}
TYPE EL1088_78E8D3DD EXTENDS EtcSlaveTerminalBase_947E5A46 :
STRUCT
	{attribute addProperty Name "Channel_1"}
	Channel_1 : Channel_830843C1;
	{attribute addProperty Name "Channel_2"}
	Channel_2 : Channel_830843C1;
	{attribute addProperty Name "Channel_3"}
	Channel_3 : Channel_830843C1;
	{attribute addProperty Name "Channel_4"}
	Channel_4 : Channel_830843C1;
	{attribute addProperty Name "Channel_5"}
	Channel_5 : Channel_830843C1;
	{attribute addProperty Name "Channel_6"}
	Channel_6 : Channel_830843C1;
	{attribute addProperty Name "Channel_7"}
	Channel_7 : Channel_830843C1;
	{attribute addProperty Name "Channel_8"}
	Channel_8 : Channel_830843C1;
	{attribute addProperty Name "WcState"}
	WcState : WcState_9091E0EB;
	{attribute addProperty Name "InfoData"}
	InfoData : InfoData_6F19DB2B;
END_STRUCT
END_TYPE

// ---- DUTs/IO/Boxes/EL1094_D135F8DB.TcDUT
{attribute 'GeneratedUsingTerminal: EL1094-0000-0016'}
{attribute addProperty BoxType "EL1094-0000-0016"}
{attribute addProperty Description "EL1094 4Ch. Dig. Input 24V, 10µs, negative"}
{attribute addProperty Physics "KK"}
{attribute addProperty Id "Channel_1AT %I*Channel_830843C11Channel_2AT %I*Channel_830843C11Channel_3AT %I*Channel_830843C11Channel_4AT %I*Channel_830843C11WcStateAT %I*WcState_9091E0EB2InfoDataAT %I*InfoData_6F19DB2B2"}
{attribute addProperty CRC "3509975259"}
{attribute addProperty Size "8"}
TYPE EL1094_D135F8DB EXTENDS EtcSlaveTerminalBase_947E5A46 :
STRUCT
	{attribute addProperty Name "Channel_1"}
	Channel_1 : Channel_830843C1;
	{attribute addProperty Name "Channel_2"}
	Channel_2 : Channel_830843C1;
	{attribute addProperty Name "Channel_3"}
	Channel_3 : Channel_830843C1;
	{attribute addProperty Name "Channel_4"}
	Channel_4 : Channel_830843C1;
	{attribute addProperty Name "WcState"}
	WcState : WcState_9091E0EB;
	{attribute addProperty Name "InfoData"}
	InfoData : InfoData_6F19DB2B;
END_STRUCT
END_TYPE

// ---- DUTs/IO/Boxes/EL1098_78E8D3DD.TcDUT
{attribute 'GeneratedUsingTerminal: EL1098-0000-0016'}
{attribute addProperty BoxType "EL1098-0000-0016"}
{attribute addProperty Description "EL1098 8Ch. Dig. Input 24V, 10µs, negative"}
{attribute addProperty Physics "KK"}
{attribute addProperty Id "Channel_1AT %I*Channel_830843C11Channel_2AT %I*Channel_830843C11Channel_3AT %I*Channel_830843C11Channel_4AT %I*Channel_830843C11Channel_5AT %I*Channel_830843C11Channel_6AT %I*Channel_830843C11Channel_7AT %I*Channel_830843C11Channel_8AT %I*Channel_830843C11WcStateAT %I*WcState_9091E0EB2InfoDataAT %I*InfoData_6F19DB2B2"}
{attribute addProperty CRC "2028524509"}
{attribute addProperty Size "12"}
TYPE EL1098_78E8D3DD EXTENDS EtcSlaveTerminalBase_947E5A46 :
STRUCT
	{attribute addProperty Name "Channel_1"}
	Channel_1 : Channel_830843C1;
	{attribute addProperty Name "Channel_2"}
	Channel_2 : Channel_830843C1;
	{attribute addProperty Name "Channel_3"}
	Channel_3 : Channel_830843C1;
	{attribute addProperty Name "Channel_4"}
	Channel_4 : Channel_830843C1;
	{attribute addProperty Name "Channel_5"}
	Channel_5 : Channel_830843C1;
	{attribute addProperty Name "Channel_6"}
	Channel_6 : Channel_830843C1;
	{attribute addProperty Name "Channel_7"}
	Channel_7 : Channel_830843C1;
	{attribute addProperty Name "Channel_8"}
	Channel_8 : Channel_830843C1;
	{attribute addProperty Name "WcState"}
	WcState : WcState_9091E0EB;
	{attribute addProperty Name "InfoData"}
	InfoData : InfoData_6F19DB2B;
END_STRUCT
END_TYPE

// ---- DUTs/IO/Boxes/EL1104_D135F8DB.TcDUT
{attribute 'GeneratedUsingTerminal: EL1104-0000-0016'}
{attribute addProperty BoxType "EL1104-0000-0016"}
{attribute addProperty Description "EL1104 4Ch. Dig. Input 24V, 3ms, Sensor Power"}
{attribute addProperty Physics "KK"}
{attribute addProperty Id "Channel_1AT %I*Channel_830843C11Channel_2AT %I*Channel_830843C11Channel_3AT %I*Channel_830843C11Channel_4AT %I*Channel_830843C11WcStateAT %I*WcState_9091E0EB2InfoDataAT %I*InfoData_6F19DB2B2"}
{attribute addProperty CRC "3509975259"}
{attribute addProperty Size "8"}
TYPE EL1104_D135F8DB EXTENDS EtcSlaveTerminalBase_947E5A46 :
STRUCT
	{attribute addProperty Name "Channel_1"}
	Channel_1 : Channel_830843C1;
	{attribute addProperty Name "Channel_2"}
	Channel_2 : Channel_830843C1;
	{attribute addProperty Name "Channel_3"}
	Channel_3 : Channel_830843C1;
	{attribute addProperty Name "Channel_4"}
	Channel_4 : Channel_830843C1;
	{attribute addProperty Name "WcState"}
	WcState : WcState_9091E0EB;
	{attribute addProperty Name "InfoData"}
	InfoData : InfoData_6F19DB2B;
END_STRUCT
END_TYPE

// ---- DUTs/IO/Boxes/EL1114_D135F8DB.TcDUT
{attribute 'GeneratedUsingTerminal: EL1114-0000-0016'}
{attribute addProperty BoxType "EL1114-0000-0016"}
{attribute addProperty Description "EL1114 4Ch. Dig. Input 24V, 10µs, Sensor Power"}
{attribute addProperty Physics "KK"}
{attribute addProperty Id "Channel_1AT %I*Channel_830843C11Channel_2AT %I*Channel_830843C11Channel_3AT %I*Channel_830843C11Channel_4AT %I*Channel_830843C11WcStateAT %I*WcState_9091E0EB2InfoDataAT %I*InfoData_6F19DB2B2"}
{attribute addProperty CRC "3509975259"}
{attribute addProperty Size "8"}
TYPE EL1114_D135F8DB EXTENDS EtcSlaveTerminalBase_947E5A46 :
STRUCT
	{attribute addProperty Name "Channel_1"}
	Channel_1 : Channel_830843C1;
	{attribute addProperty Name "Channel_2"}
	Channel_2 : Channel_830843C1;
	{attribute addProperty Name "Channel_3"}
	Channel_3 : Channel_830843C1;
	{attribute addProperty Name "Channel_4"}
	Channel_4 : Channel_830843C1;
	{attribute addProperty Name "WcState"}
	WcState : WcState_9091E0EB;
	{attribute addProperty Name "InfoData"}
	InfoData : InfoData_6F19DB2B;
END_STRUCT
END_TYPE

// ---- DUTs/IO/Boxes/EL1124_D135F8DB.TcDUT
{attribute 'GeneratedUsingTerminal: EL1124-0000-0016'}
{attribute addProperty BoxType "EL1124-0000-0016"}
{attribute addProperty Description "EL1124 4Ch. Dig. Input 5V, 10µs, Sensor Power"}
{attribute addProperty Physics "KK"}
{attribute addProperty Id "Channel_1AT %I*Channel_830843C11Channel_2AT %I*Channel_830843C11Channel_3AT %I*Channel_830843C11Channel_4AT %I*Channel_830843C11WcStateAT %I*WcState_9091E0EB2InfoDataAT %I*InfoData_6F19DB2B2"}
{attribute addProperty CRC "3509975259"}
{attribute addProperty Size "8"}
TYPE EL1124_D135F8DB EXTENDS EtcSlaveTerminalBase_947E5A46 :
STRUCT
	{attribute addProperty Name "Channel_1"}
	Channel_1 : Channel_830843C1;
	{attribute addProperty Name "Channel_2"}
	Channel_2 : Channel_830843C1;
	{attribute addProperty Name "Channel_3"}
	Channel_3 : Channel_830843C1;
	{attribute addProperty Name "Channel_4"}
	Channel_4 : Channel_830843C1;
	{attribute addProperty Name "WcState"}
	WcState : WcState_9091E0EB;
	{attribute addProperty Name "InfoData"}
	InfoData : InfoData_6F19DB2B;
END_STRUCT
END_TYPE

// ---- DUTs/IO/Boxes/EL1134_D135F8DB.TcDUT
{attribute 'GeneratedUsingTerminal: EL1134-0000-0016'}
{attribute addProperty BoxType "EL1134-0000-0016"}
{attribute addProperty Description "EL1134 4Ch. Dig. Input 48V, 10µs, Sensor Power"}
{attribute addProperty Physics "KK"}
{attribute addProperty Id "Channel_1AT %I*Channel_830843C11Channel_2AT %I*Channel_830843C11Channel_3AT %I*Channel_830843C11Channel_4AT %I*Channel_830843C11WcStateAT %I*WcState_9091E0EB2InfoDataAT %I*InfoData_6F19DB2B2"}
{attribute addProperty CRC "3509975259"}
{attribute addProperty Size "8"}
TYPE EL1134_D135F8DB EXTENDS EtcSlaveTerminalBase_947E5A46 :
STRUCT
	{attribute addProperty Name "Channel_1"}
	Channel_1 : Channel_830843C1;
	{attribute addProperty Name "Channel_2"}
	Channel_2 : Channel_830843C1;
	{attribute addProperty Name "Channel_3"}
	Channel_3 : Channel_830843C1;
	{attribute addProperty Name "Channel_4"}
	Channel_4 : Channel_830843C1;
	{attribute addProperty Name "WcState"}
	WcState : WcState_9091E0EB;
	{attribute addProperty Name "InfoData"}
	InfoData : InfoData_6F19DB2B;
END_STRUCT
END_TYPE

// ---- DUTs/IO/Boxes/EL1144_D135F8DB.TcDUT
{attribute 'GeneratedUsingTerminal: EL1144-0000-0016'}
{attribute addProperty BoxType "EL1144-0000-0016"}
{attribute addProperty Description "EL1144 4Ch. Dig. Input 12V, 10µs, Sensor Power"}
{attribute addProperty Physics "KK"}
{attribute addProperty Id "Channel_1AT %I*Channel_830843C11Channel_2AT %I*Channel_830843C11Channel_3AT %I*Channel_830843C11Channel_4AT %I*Channel_830843C11WcStateAT %I*WcState_9091E0EB2InfoDataAT %I*InfoData_6F19DB2B2"}
{attribute addProperty CRC "3509975259"}
{attribute addProperty Size "8"}
TYPE EL1144_D135F8DB EXTENDS EtcSlaveTerminalBase_947E5A46 :
STRUCT
	{attribute addProperty Name "Channel_1"}
	Channel_1 : Channel_830843C1;
	{attribute addProperty Name "Channel_2"}
	Channel_2 : Channel_830843C1;
	{attribute addProperty Name "Channel_3"}
	Channel_3 : Channel_830843C1;
	{attribute addProperty Name "Channel_4"}
	Channel_4 : Channel_830843C1;
	{attribute addProperty Name "WcState"}
	WcState : WcState_9091E0EB;
	{attribute addProperty Name "InfoData"}
	InfoData : InfoData_6F19DB2B;
END_STRUCT
END_TYPE

// ---- DUTs/IO/Boxes/EL1202_02444DCB.TcDUT
{attribute 'GeneratedUsingTerminal: EL1202-0000-0016'}
{attribute addProperty BoxType "EL1202-0000-0016"}
{attribute addProperty Description "EL1202 2Ch. Fast Dig. Input 24V, 1µs"}
{attribute addProperty Physics "KK"}
{attribute addProperty Id "Channel_1AT %I*Channel_830843C11Channel_2AT %I*Channel_830843C11WcStateAT %I*WcState_9091E0EB2InfoDataAT %I*InfoData_6F19DB2B2"}
{attribute addProperty CRC "38030795"}
{attribute addProperty Size "6"}
TYPE EL1202_02444DCB EXTENDS EtcSlaveTerminalBase_947E5A46 :
STRUCT
	{attribute addProperty Name "Channel_1"}
	Channel_1 : Channel_830843C1;
	{attribute addProperty Name "Channel_2"}
	Channel_2 : Channel_830843C1;
	{attribute addProperty Name "WcState"}
	WcState : WcState_9091E0EB;
	{attribute addProperty Name "InfoData"}
	InfoData : InfoData_6F19DB2B;
END_STRUCT
END_TYPE

// ---- DUTs/IO/Boxes/EL1202_647E4607.TcDUT
{attribute 'GeneratedUsingTerminal: EL1202-0100-0016'}
{attribute addProperty BoxType "EL1202-0100-0016"}
{attribute addProperty Description "EL1202-0100 2Ch. Fast Dig. Input 24V, 1µs, DC Latch"}
{attribute addProperty Physics "KK"}
{attribute addProperty Id "Channel_1AT %I*Channel_830843C11Channel_2AT %I*Channel_830843C11ReservedEMPTY_STRUCTURE0DCAT %I*DC_1A6E66258WcStateAT %I*WcState_9091E0EB2InfoDataAT %I*InfoData_A7436BC610"}
{attribute addProperty CRC "1685997063"}
{attribute addProperty Size "22"}
TYPE EL1202_647E4607 EXTENDS EtcSlaveTerminalBase_947E5A46 :
STRUCT
	{attribute addProperty Name "Channel_1"}
	Channel_1 : Channel_830843C1;
	{attribute addProperty Name "Channel_2"}
	Channel_2 : Channel_830843C1;
	{attribute addProperty Name "Reserved"}
	Reserved : EMPTY_STRUCTURE;
	{attribute addProperty Name "DC"}
	DC : DC_1A6E6625;
	{attribute addProperty Name "WcState"}
	WcState : WcState_9091E0EB;
	{attribute addProperty Name "InfoData"}
	InfoData : InfoData_A7436BC6;
END_STRUCT
END_TYPE

// ---- DUTs/IO/Boxes/EL1252_0C2D47B4.TcDUT
{attribute 'GeneratedUsingTerminal: EL1252-0000-0017'}
{attribute addProperty BoxType "EL1252-0000-0017"}
{attribute addProperty Description "EL1252 2Ch. Fast Dig. Input 24V, 1µs, DC Latch"}
{attribute addProperty Physics "KK"}
{attribute addProperty Id "LatchAT %I*Latch_8E41329534Channel_0AT %I*Channel_830843C11Channel_1AT %I*Channel_830843C11ReservedEMPTY_STRUCTURE0WcStateAT %I*WcState_9091E0EB2InfoDataAT %I*InfoData_A7436BC610"}
{attribute addProperty CRC "204294068"}
{attribute addProperty Size "48"}
TYPE EL1252_0C2D47B4 EXTENDS EtcSlaveTerminalBase_947E5A46 :
STRUCT
	{attribute addProperty Name "Latch"}
	Latch : Latch_8E413295;
	{attribute addProperty Name "Channel_0"}
	Channel_0 : Channel_830843C1;
	{attribute addProperty Name "Channel_1"}
	Channel_1 : Channel_830843C1;
	{attribute addProperty Name "Reserved"}
	Reserved : EMPTY_STRUCTURE;
	{attribute addProperty Name "WcState"}
	WcState : WcState_9091E0EB;
	{attribute addProperty Name "InfoData"}
	InfoData : InfoData_A7436BC6;
END_STRUCT
END_TYPE

// ---- DUTs/IO/Boxes/EL1252_934A18FC.TcDUT
{attribute 'GeneratedUsingTerminal: EL1252-0000-0018'}
{attribute addProperty BoxType "EL1252-0000-0018"}
{attribute addProperty Description "EL1252 2Ch. Fast Dig. Input 24V, 1µs, DC Latch"}
{attribute addProperty Physics "KK"}
{attribute addProperty Id "Channel_1AT %I*Channel_830843C11Channel_2AT %I*Channel_830843C11ReservedEMPTY_STRUCTURE0LatchAT %I*Latch_39BD7C7C34WcStateAT %I*WcState_9091E0EB2InfoDataAT %I*InfoData_A7436BC610"}
{attribute addProperty CRC "2471106812"}
{attribute addProperty Size "48"}
TYPE EL1252_934A18FC EXTENDS EtcSlaveTerminalBase_947E5A46 :
STRUCT
	{attribute addProperty Name "Channel_1"}
	Channel_1 : Channel_830843C1;
	{attribute addProperty Name "Channel_2"}
	Channel_2 : Channel_830843C1;
	{attribute addProperty Name "Reserved"}
	Reserved : EMPTY_STRUCTURE;
	{attribute addProperty Name "Latch"}
	Latch : Latch_39BD7C7C;
	{attribute addProperty Name "WcState"}
	WcState : WcState_9091E0EB;
	{attribute addProperty Name "InfoData"}
	InfoData : InfoData_A7436BC6;
END_STRUCT
END_TYPE

// ---- DUTs/IO/Boxes/EL1254_D5E6FA5F.TcDUT
{attribute 'GeneratedUsingTerminal: EL1254--0000'}
{attribute addProperty BoxType "EL1254--0000"}
{attribute addProperty Description "EL1254 4Ch. Fast Dig. Input 24V, 1µs, DC Latch"}
{attribute addProperty Physics "KK"}
{attribute addProperty Id "Channel_1AT %I*Channel_830843C11Channel_2AT %I*Channel_830843C11Channel_3AT %I*Channel_830843C11Channel_4AT %I*Channel_830843C11ReservedEMPTY_STRUCTURE0LatchAT %I*Latch_0465F91668WcStateAT %I*WcState_9091E0EB2InfoDataAT %I*InfoData_A7436BC610"}
{attribute addProperty CRC "3588684383"}
{attribute addProperty Size "84"}
TYPE EL1254_D5E6FA5F EXTENDS EtcSlaveTerminalBase_947E5A46 :
STRUCT
	{attribute addProperty Name "Channel_1"}
	Channel_1 : Channel_830843C1;
	{attribute addProperty Name "Channel_2"}
	Channel_2 : Channel_830843C1;
	{attribute addProperty Name "Channel_3"}
	Channel_3 : Channel_830843C1;
	{attribute addProperty Name "Channel_4"}
	Channel_4 : Channel_830843C1;
	{attribute addProperty Name "Reserved"}
	Reserved : EMPTY_STRUCTURE;
	{attribute addProperty Name "Latch"}
	Latch : Latch_0465F916;
	{attribute addProperty Name "WcState"}
	WcState : WcState_9091E0EB;
	{attribute addProperty Name "InfoData"}
	InfoData : InfoData_A7436BC6;
END_STRUCT
END_TYPE

// ---- DUTs/IO/Boxes/EL1262_0FA571DE.TcDUT
{attribute 'GeneratedUsingTerminal: EL1262-0000-0002'}
{attribute addProperty BoxType "EL1262-0000-0002"}
{attribute addProperty Description "EL1262 2Ch. Dig. Input 24V, 1µs, DC Oversample"}
{attribute addProperty Physics "KK"}
{attribute addProperty Id "Ch1_CycleCountAT %I*Ch1_CycleCount_9DBE2BC52Ch1_Input_0AT %I*Ch1_Input_FFC4CE241Ch1_Input_1AT %I*Ch1_Input_FFC4CE241Ch1_Input_2AT %I*Ch1_Input_FFC4CE241Ch1_Input_3AT %I*Ch1_Input_FFC4CE241Ch1_Input_4AT %I*Ch1_Input_FFC4CE241Ch1_Input_5AT %I*Ch1_Input_FFC4CE241Ch1_Input_6AT %I*Ch1_Input_FFC4CE241Ch1_Input_7AT %I*Ch1_Input_FFC4CE241Ch1_Input_8AT %I*Ch1_Input_FFC4CE241Ch1_Input_9AT %I*Ch1_Input_FFC4CE241GapAT %I*EMPTY_STRUCTURE0Ch2_CycleCountAT %I*Ch2_CycleCount_976A51B52Ch2_Input_0AT %I*Ch2_Input_78ADA90C1Ch2_Input_1AT %I*Ch2_Input_78ADA90C1Ch2_Input_2AT %I*Ch2_Input_78ADA90C1Ch2_Input_3AT %I*Ch2_Input_78ADA90C1Ch2_Input_4AT %I*Ch2_Input_78ADA90C1Ch2_Input_5AT %I*Ch2_Input_78ADA90C1Ch2_Input_6AT %I*Ch2_Input_78ADA90C1Ch2_Input_7AT %I*Ch2_Input_78ADA90C1Ch2_Input_8AT %I*Ch2_Input_78ADA90C1Ch2_Input_9AT %I*Ch2_Input_78ADA90C1Gap_1AT %I*EMPTY_STRUCTURE0NextSync1TimeAT %I*NextSync1Time_EE185E174WcStateAT %I*WcState_9091E0EB2InfoDataAT %I*InfoData_A7436BC610"}
{attribute addProperty CRC "262500830"}
{attribute addProperty Size "40"}
TYPE EL1262_0FA571DE EXTENDS EtcSlaveTerminalBase_947E5A46 :
STRUCT
	{attribute addProperty Name "Ch1_CycleCount"}
	Ch1_CycleCount : Ch1_CycleCount_9DBE2BC5;
	{attribute addProperty Name "Ch1_Input_0"}
	Ch1_Input_0 : Ch1_Input_FFC4CE24;
	{attribute addProperty Name "Ch1_Input_1"}
	Ch1_Input_1 : Ch1_Input_FFC4CE24;
	{attribute addProperty Name "Ch1_Input_2"}
	Ch1_Input_2 : Ch1_Input_FFC4CE24;
	{attribute addProperty Name "Ch1_Input_3"}
	Ch1_Input_3 : Ch1_Input_FFC4CE24;
	{attribute addProperty Name "Ch1_Input_4"}
	Ch1_Input_4 : Ch1_Input_FFC4CE24;
	{attribute addProperty Name "Ch1_Input_5"}
	Ch1_Input_5 : Ch1_Input_FFC4CE24;
	{attribute addProperty Name "Ch1_Input_6"}
	Ch1_Input_6 : Ch1_Input_FFC4CE24;
	{attribute addProperty Name "Ch1_Input_7"}
	Ch1_Input_7 : Ch1_Input_FFC4CE24;
	{attribute addProperty Name "Ch1_Input_8"}
	Ch1_Input_8 : Ch1_Input_FFC4CE24;
	{attribute addProperty Name "Ch1_Input_9"}
	Ch1_Input_9 : Ch1_Input_FFC4CE24;
	{attribute addProperty Name "Gap"}
	Gap : EMPTY_STRUCTURE;
	{attribute addProperty Name "Ch2_CycleCount"}
	Ch2_CycleCount : Ch2_CycleCount_976A51B5;
	{attribute addProperty Name "Ch2_Input_0"}
	Ch2_Input_0 : Ch2_Input_78ADA90C;
	{attribute addProperty Name "Ch2_Input_1"}
	Ch2_Input_1 : Ch2_Input_78ADA90C;
	{attribute addProperty Name "Ch2_Input_2"}
	Ch2_Input_2 : Ch2_Input_78ADA90C;
	{attribute addProperty Name "Ch2_Input_3"}
	Ch2_Input_3 : Ch2_Input_78ADA90C;
	{attribute addProperty Name "Ch2_Input_4"}
	Ch2_Input_4 : Ch2_Input_78ADA90C;
	{attribute addProperty Name "Ch2_Input_5"}
	Ch2_Input_5 : Ch2_Input_78ADA90C;
	{attribute addProperty Name "Ch2_Input_6"}
	Ch2_Input_6 : Ch2_Input_78ADA90C;
	{attribute addProperty Name "Ch2_Input_7"}
	Ch2_Input_7 : Ch2_Input_78ADA90C;
	{attribute addProperty Name "Ch2_Input_8"}
	Ch2_Input_8 : Ch2_Input_78ADA90C;
	{attribute addProperty Name "Ch2_Input_9"}
	Ch2_Input_9 : Ch2_Input_78ADA90C;
	{attribute addProperty Name "Gap_1"}
	Gap_1 : EMPTY_STRUCTURE;
	{attribute addProperty Name "NextSync1Time"}
	NextSync1Time : NextSync1Time_EE185E17;
	{attribute addProperty Name "WcState"}
	WcState : WcState_9091E0EB;
	{attribute addProperty Name "InfoData"}
	InfoData : InfoData_A7436BC6;
END_STRUCT
END_TYPE

// ---- DUTs/IO/Boxes/EL1258_733F03F2.TcDUT
{attribute 'GeneratedUsingTerminal: EL1258-0000-0016'}
{attribute addProperty BoxType "EL1258-0000-0016"}
{attribute addProperty Description "EL1258 8Ch. Dig Input 24V with Multi-Time-Stamp"}
{attribute addProperty Physics "KK"}
{attribute addProperty Id "MTI_Inputs_10x_Channel_1AT %I*MTI_Inputs_10x_Channel_C3ED30FD56MTI_Inputs_10x_Channel_2AT %I*MTI_Inputs_10x_Channel_C3ED30FD56MTI_Inputs_10x_Channel_3AT %I*MTI_Inputs_10x_Channel_C3ED30FD56MTI_Inputs_10x_Channel_4AT %I*MTI_Inputs_10x_Channel_C3ED30FD56MTI_Inputs_10x_Channel_5AT %I*MTI_Inputs_10x_Channel_C3ED30FD56MTI_Inputs_10x_Channel_6AT %I*MTI_Inputs_10x_Channel_C3ED30FD56MTI_Inputs_10x_Channel_7AT %I*MTI_Inputs_10x_Channel_C3ED30FD56MTI_Inputs_10x_Channel_8AT %I*MTI_Inputs_10x_Channel_C3ED30FD56MTI_Outputs_Channel_1AT %Q*MTI_Outputs_Channel_0F1028A12MTI_Outputs_Channel_2AT %Q*MTI_Outputs_Channel_0F1028A12MTI_Outputs_Channel_3AT %Q*MTI_Outputs_Channel_0F1028A12MTI_Outputs_Channel_4AT %Q*MTI_Outputs_Channel_0F1028A12MTI_Outputs_Channel_5AT %Q*MTI_Outputs_Channel_0F1028A12MTI_Outputs_Channel_6AT %Q*MTI_Outputs_Channel_0F1028A12MTI_Outputs_Channel_7AT %Q*MTI_Outputs_Channel_0F1028A12MTI_Outputs_Channel_8AT %Q*MTI_Outputs_Channel_0F1028A12WcStateAT %I*WcState_9091E0EB2InfoDataAT %I*InfoData_BEF6B88E18"}
{attribute addProperty CRC "1933509618"}
{attribute addProperty Size "484"}
TYPE EL1258_733F03F2 EXTENDS EtcSlaveTerminalBase_947E5A46 :
STRUCT
	{attribute addProperty Name "MTI_Inputs_10x_Channel_1"}
	MTI_Inputs_10x_Channel_1 : MTI_Inputs_10x_Channel_C3ED30FD;
	{attribute addProperty Name "MTI_Inputs_10x_Channel_2"}
	MTI_Inputs_10x_Channel_2 : MTI_Inputs_10x_Channel_C3ED30FD;
	{attribute addProperty Name "MTI_Inputs_10x_Channel_3"}
	MTI_Inputs_10x_Channel_3 : MTI_Inputs_10x_Channel_C3ED30FD;
	{attribute addProperty Name "MTI_Inputs_10x_Channel_4"}
	MTI_Inputs_10x_Channel_4 : MTI_Inputs_10x_Channel_C3ED30FD;
	{attribute addProperty Name "MTI_Inputs_10x_Channel_5"}
	MTI_Inputs_10x_Channel_5 : MTI_Inputs_10x_Channel_C3ED30FD;
	{attribute addProperty Name "MTI_Inputs_10x_Channel_6"}
	MTI_Inputs_10x_Channel_6 : MTI_Inputs_10x_Channel_C3ED30FD;
	{attribute addProperty Name "MTI_Inputs_10x_Channel_7"}
	MTI_Inputs_10x_Channel_7 : MTI_Inputs_10x_Channel_C3ED30FD;
	{attribute addProperty Name "MTI_Inputs_10x_Channel_8"}
	MTI_Inputs_10x_Channel_8 : MTI_Inputs_10x_Channel_C3ED30FD;
	{attribute addProperty Name "MTI_Outputs_Channel_1"}
	MTI_Outputs_Channel_1 : MTI_Outputs_Channel_0F1028A1;
	{attribute addProperty Name "MTI_Outputs_Channel_2"}
	MTI_Outputs_Channel_2 : MTI_Outputs_Channel_0F1028A1;
	{attribute addProperty Name "MTI_Outputs_Channel_3"}
	MTI_Outputs_Channel_3 : MTI_Outputs_Channel_0F1028A1;
	{attribute addProperty Name "MTI_Outputs_Channel_4"}
	MTI_Outputs_Channel_4 : MTI_Outputs_Channel_0F1028A1;
	{attribute addProperty Name "MTI_Outputs_Channel_5"}
	MTI_Outputs_Channel_5 : MTI_Outputs_Channel_0F1028A1;
	{attribute addProperty Name "MTI_Outputs_Channel_6"}
	MTI_Outputs_Channel_6 : MTI_Outputs_Channel_0F1028A1;
	{attribute addProperty Name "MTI_Outputs_Channel_7"}
	MTI_Outputs_Channel_7 : MTI_Outputs_Channel_0F1028A1;
	{attribute addProperty Name "MTI_Outputs_Channel_8"}
	MTI_Outputs_Channel_8 : MTI_Outputs_Channel_0F1028A1;
	{attribute addProperty Name "WcState"}
	WcState : WcState_9091E0EB;
	{attribute addProperty Name "InfoData"}
	InfoData : InfoData_BEF6B88E;
END_STRUCT
END_TYPE

// ---- DUTs/IO/Boxes/EL1258_699E7002.TcDUT
{attribute 'GeneratedUsingTerminal: EL1258-0010-0017'}
{attribute addProperty BoxType "EL1258-0010-0017"}
{attribute addProperty Description "EL1258-0010 8Ch. Dig Input 24V with Multi-Time-Stamp, ground switching"}
{attribute addProperty Physics "KK"}
{attribute addProperty Id "MTI_Inputs_1x_Channel_1AT %I*MTI_Inputs_1x_Channel_CC1B212F11MTI_Inputs_1x_Channel_2AT %I*MTI_Inputs_1x_Channel_CC1B212F11MTI_Inputs_1x_Channel_3AT %I*MTI_Inputs_1x_Channel_CC1B212F11MTI_Inputs_1x_Channel_4AT %I*MTI_Inputs_1x_Channel_CC1B212F11MTI_Inputs_1x_Channel_5AT %I*MTI_Inputs_1x_Channel_CC1B212F11MTI_Inputs_1x_Channel_6AT %I*MTI_Inputs_1x_Channel_CC1B212F11MTI_Inputs_1x_Channel_7AT %I*MTI_Inputs_1x_Channel_CC1B212F11MTI_Inputs_1x_Channel_8AT %I*MTI_Inputs_1x_Channel_CC1B212F11MTI_Outputs_Channel_1AT %Q*MTI_Outputs_Channel_0F1028A12MTI_Outputs_Channel_2AT %Q*MTI_Outputs_Channel_0F1028A12MTI_Outputs_Channel_3AT %Q*MTI_Outputs_Channel_0F1028A12MTI_Outputs_Channel_4AT %Q*MTI_Outputs_Channel_0F1028A12MTI_Outputs_Channel_5AT %Q*MTI_Outputs_Channel_0F1028A12MTI_Outputs_Channel_6AT %Q*MTI_Outputs_Channel_0F1028A12MTI_Outputs_Channel_7AT %Q*MTI_Outputs_Channel_0F1028A12MTI_Outputs_Channel_8AT %Q*MTI_Outputs_Channel_0F1028A12WcStateAT %I*WcState_9091E0EB2InfoDataAT %I*InfoData_BEF6B88E18"}
{attribute addProperty CRC "1771991042"}
{attribute addProperty Size "124"}
TYPE EL1258_699E7002 EXTENDS EtcSlaveTerminalBase_947E5A46 :
STRUCT
	{attribute addProperty Name "MTI_Inputs_1x_Channel_1"}
	MTI_Inputs_1x_Channel_1 : MTI_Inputs_1x_Channel_CC1B212F;
	{attribute addProperty Name "MTI_Inputs_1x_Channel_2"}
	MTI_Inputs_1x_Channel_2 : MTI_Inputs_1x_Channel_CC1B212F;
	{attribute addProperty Name "MTI_Inputs_1x_Channel_3"}
	MTI_Inputs_1x_Channel_3 : MTI_Inputs_1x_Channel_CC1B212F;
	{attribute addProperty Name "MTI_Inputs_1x_Channel_4"}
	MTI_Inputs_1x_Channel_4 : MTI_Inputs_1x_Channel_CC1B212F;
	{attribute addProperty Name "MTI_Inputs_1x_Channel_5"}
	MTI_Inputs_1x_Channel_5 : MTI_Inputs_1x_Channel_CC1B212F;
	{attribute addProperty Name "MTI_Inputs_1x_Channel_6"}
	MTI_Inputs_1x_Channel_6 : MTI_Inputs_1x_Channel_CC1B212F;
	{attribute addProperty Name "MTI_Inputs_1x_Channel_7"}
	MTI_Inputs_1x_Channel_7 : MTI_Inputs_1x_Channel_CC1B212F;
	{attribute addProperty Name "MTI_Inputs_1x_Channel_8"}
	MTI_Inputs_1x_Channel_8 : MTI_Inputs_1x_Channel_CC1B212F;
	{attribute addProperty Name "MTI_Outputs_Channel_1"}
	MTI_Outputs_Channel_1 : MTI_Outputs_Channel_0F1028A1;
	{attribute addProperty Name "MTI_Outputs_Channel_2"}
	MTI_Outputs_Channel_2 : MTI_Outputs_Channel_0F1028A1;
	{attribute addProperty Name "MTI_Outputs_Channel_3"}
	MTI_Outputs_Channel_3 : MTI_Outputs_Channel_0F1028A1;
	{attribute addProperty Name "MTI_Outputs_Channel_4"}
	MTI_Outputs_Channel_4 : MTI_Outputs_Channel_0F1028A1;
	{attribute addProperty Name "MTI_Outputs_Channel_5"}
	MTI_Outputs_Channel_5 : MTI_Outputs_Channel_0F1028A1;
	{attribute addProperty Name "MTI_Outputs_Channel_6"}
	MTI_Outputs_Channel_6 : MTI_Outputs_Channel_0F1028A1;
	{attribute addProperty Name "MTI_Outputs_Channel_7"}
	MTI_Outputs_Channel_7 : MTI_Outputs_Channel_0F1028A1;
	{attribute addProperty Name "MTI_Outputs_Channel_8"}
	MTI_Outputs_Channel_8 : MTI_Outputs_Channel_0F1028A1;
	{attribute addProperty Name "WcState"}
	WcState : WcState_9091E0EB;
	{attribute addProperty Name "InfoData"}
	InfoData : InfoData_BEF6B88E;
END_STRUCT
END_TYPE

// ---- DUTs/IO/Boxes/EL1259_5165368D.TcDUT
{attribute 'GeneratedUsingTerminal: EL1259-0000-0016'}
{attribute addProperty BoxType "EL1259-0000-0016"}
{attribute addProperty Description "EL1259 8Ch. Dig Input 24V/8Ch. Dig. Output 24V with Multi-Time-Stamp"}
{attribute addProperty Physics "KK"}
{attribute addProperty Id "MTO_Inputs_Channel_1AT %I*MTO_Inputs_Channel_53C09E8B6MTO_Inputs_Channel_2AT %I*MTO_Inputs_Channel_53C09E8B6MTO_Inputs_Channel_3AT %I*MTO_Inputs_Channel_53C09E8B6MTO_Inputs_Channel_4AT %I*MTO_Inputs_Channel_53C09E8B6MTO_Inputs_Channel_5AT %I*MTO_Inputs_Channel_53C09E8B6MTO_Inputs_Channel_6AT %I*MTO_Inputs_Channel_53C09E8B6MTO_Inputs_Channel_7AT %I*MTO_Inputs_Channel_53C09E8B6MTO_Inputs_Channel_8AT %I*MTO_Inputs_Channel_53C09E8B6MTI_Inputs_10x_Channel_1AT %I*MTI_Inputs_10x_Channel_C3ED30FD56MTI_Inputs_10x_Channel_2AT %I*MTI_Inputs_10x_Channel_C3ED30FD56MTI_Inputs_10x_Channel_3AT %I*MTI_Inputs_10x_Channel_C3ED30FD56MTI_Inputs_10x_Channel_4AT %I*MTI_Inputs_10x_Channel_C3ED30FD56MTI_Inputs_10x_Channel_5AT %I*MTI_Inputs_10x_Channel_C3ED30FD56MTI_Inputs_10x_Channel_6AT %I*MTI_Inputs_10x_Channel_C3ED30FD56MTI_Inputs_10x_Channel_7AT %I*MTI_Inputs_10x_Channel_C3ED30FD56MTI_Inputs_10x_Channel_8AT %I*MTI_Inputs_10x_Channel_C3ED30FD56MTO_Outputs_10x_Channel_1AT %Q*MTO_Outputs_10x_Channel_232E011755MTO_Outputs_10x_Channel_2AT %Q*MTO_Outputs_10x_Channel_232E011755MTO_Outputs_10x_Channel_3AT %Q*MTO_Outputs_10x_Channel_232E011755MTO_Outputs_10x_Channel_4AT %Q*MTO_Outputs_10x_Channel_232E011755MTO_Outputs_10x_Channel_5AT %Q*MTO_Outputs_10x_Channel_232E011755MTO_Outputs_10x_Channel_6AT %Q*MTO_Outputs_10x_Channel_232E011755MTO_Outputs_10x_Channel_7AT %Q*MTO_Outputs_10x_Channel_232E011755MTO_Outputs_10x_Channel_8AT %Q*MTO_Outputs_10x_Channel_232E011755MTI_Outputs_Channel_1AT %Q*MTI_Outputs_Channel_0F1028A12MTI_Outputs_Channel_2AT %Q*MTI_Outputs_Channel_0F1028A12MTI_Outputs_Channel_3AT %Q*MTI_Outputs_Channel_0F1028A12MTI_Outputs_Channel_4AT %Q*MTI_Outputs_Channel_0F1028A12MTI_Outputs_Channel_5AT %Q*MTI_Outputs_Channel_0F1028A12MTI_Outputs_Channel_6AT %Q*MTI_Outputs_Channel_0F1028A12MTI_Outputs_Channel_7AT %Q*MTI_Outputs_Channel_0F1028A12MTI_Outputs_Channel_8AT %Q*MTI_Outputs_Channel_0F1028A12WcStateAT %I*WcState_9091E0EB2InfoDataAT %I*InfoData_BEF6B88E18"}
{attribute addProperty CRC "1365587597"}
{attribute addProperty Size "972"}
TYPE EL1259_5165368D EXTENDS EtcSlaveTerminalBase_947E5A46 :
STRUCT
	{attribute addProperty Name "MTO_Inputs_Channel_1"}
	MTO_Inputs_Channel_1 : MTO_Inputs_Channel_53C09E8B;
	{attribute addProperty Name "MTO_Inputs_Channel_2"}
	MTO_Inputs_Channel_2 : MTO_Inputs_Channel_53C09E8B;
	{attribute addProperty Name "MTO_Inputs_Channel_3"}
	MTO_Inputs_Channel_3 : MTO_Inputs_Channel_53C09E8B;
	{attribute addProperty Name "MTO_Inputs_Channel_4"}
	MTO_Inputs_Channel_4 : MTO_Inputs_Channel_53C09E8B;
	{attribute addProperty Name "MTO_Inputs_Channel_5"}
	MTO_Inputs_Channel_5 : MTO_Inputs_Channel_53C09E8B;
	{attribute addProperty Name "MTO_Inputs_Channel_6"}
	MTO_Inputs_Channel_6 : MTO_Inputs_Channel_53C09E8B;
	{attribute addProperty Name "MTO_Inputs_Channel_7"}
	MTO_Inputs_Channel_7 : MTO_Inputs_Channel_53C09E8B;
	{attribute addProperty Name "MTO_Inputs_Channel_8"}
	MTO_Inputs_Channel_8 : MTO_Inputs_Channel_53C09E8B;
	{attribute addProperty Name "MTI_Inputs_10x_Channel_1"}
	MTI_Inputs_10x_Channel_1 : MTI_Inputs_10x_Channel_C3ED30FD;
	{attribute addProperty Name "MTI_Inputs_10x_Channel_2"}
	MTI_Inputs_10x_Channel_2 : MTI_Inputs_10x_Channel_C3ED30FD;
	{attribute addProperty Name "MTI_Inputs_10x_Channel_3"}
	MTI_Inputs_10x_Channel_3 : MTI_Inputs_10x_Channel_C3ED30FD;
	{attribute addProperty Name "MTI_Inputs_10x_Channel_4"}
	MTI_Inputs_10x_Channel_4 : MTI_Inputs_10x_Channel_C3ED30FD;
	{attribute addProperty Name "MTI_Inputs_10x_Channel_5"}
	MTI_Inputs_10x_Channel_5 : MTI_Inputs_10x_Channel_C3ED30FD;
	{attribute addProperty Name "MTI_Inputs_10x_Channel_6"}
	MTI_Inputs_10x_Channel_6 : MTI_Inputs_10x_Channel_C3ED30FD;
	{attribute addProperty Name "MTI_Inputs_10x_Channel_7"}
	MTI_Inputs_10x_Channel_7 : MTI_Inputs_10x_Channel_C3ED30FD;
	{attribute addProperty Name "MTI_Inputs_10x_Channel_8"}
	MTI_Inputs_10x_Channel_8 : MTI_Inputs_10x_Channel_C3ED30FD;
	{attribute addProperty Name "MTO_Outputs_10x_Channel_1"}
	MTO_Outputs_10x_Channel_1 : MTO_Outputs_10x_Channel_232E0117;
	{attribute addProperty Name "MTO_Outputs_10x_Channel_2"}
	MTO_Outputs_10x_Channel_2 : MTO_Outputs_10x_Channel_232E0117;
	{attribute addProperty Name "MTO_Outputs_10x_Channel_3"}
	MTO_Outputs_10x_Channel_3 : MTO_Outputs_10x_Channel_232E0117;
	{attribute addProperty Name "MTO_Outputs_10x_Channel_4"}
	MTO_Outputs_10x_Channel_4 : MTO_Outputs_10x_Channel_232E0117;
	{attribute addProperty Name "MTO_Outputs_10x_Channel_5"}
	MTO_Outputs_10x_Channel_5 : MTO_Outputs_10x_Channel_232E0117;
	{attribute addProperty Name "MTO_Outputs_10x_Channel_6"}
	MTO_Outputs_10x_Channel_6 : MTO_Outputs_10x_Channel_232E0117;
	{attribute addProperty Name "MTO_Outputs_10x_Channel_7"}
	MTO_Outputs_10x_Channel_7 : MTO_Outputs_10x_Channel_232E0117;
	{attribute addProperty Name "MTO_Outputs_10x_Channel_8"}
	MTO_Outputs_10x_Channel_8 : MTO_Outputs_10x_Channel_232E0117;
	{attribute addProperty Name "MTI_Outputs_Channel_1"}
	MTI_Outputs_Channel_1 : MTI_Outputs_Channel_0F1028A1;
	{attribute addProperty Name "MTI_Outputs_Channel_2"}
	MTI_Outputs_Channel_2 : MTI_Outputs_Channel_0F1028A1;
	{attribute addProperty Name "MTI_Outputs_Channel_3"}
	MTI_Outputs_Channel_3 : MTI_Outputs_Channel_0F1028A1;
	{attribute addProperty Name "MTI_Outputs_Channel_4"}
	MTI_Outputs_Channel_4 : MTI_Outputs_Channel_0F1028A1;
	{attribute addProperty Name "MTI_Outputs_Channel_5"}
	MTI_Outputs_Channel_5 : MTI_Outputs_Channel_0F1028A1;
	{attribute addProperty Name "MTI_Outputs_Channel_6"}
	MTI_Outputs_Channel_6 : MTI_Outputs_Channel_0F1028A1;
	{attribute addProperty Name "MTI_Outputs_Channel_7"}
	MTI_Outputs_Channel_7 : MTI_Outputs_Channel_0F1028A1;
	{attribute addProperty Name "MTI_Outputs_Channel_8"}
	MTI_Outputs_Channel_8 : MTI_Outputs_Channel_0F1028A1;
	{attribute addProperty Name "WcState"}
	WcState : WcState_9091E0EB;
	{attribute addProperty Name "InfoData"}
	InfoData : InfoData_BEF6B88E;
END_STRUCT
END_TYPE

// ---- DUTs/IO/Boxes/EL1259_AB1DE4FC.TcDUT
{attribute 'GeneratedUsingTerminal: EL1259-0000-0017'}
{attribute addProperty BoxType "EL1259-0000-0017"}
{attribute addProperty Description "EL1259 8Ch. Dig Input 24V/8Ch. Dig. Output 24V with Multi-Time-Stamp"}
{attribute addProperty Physics "KK"}
{attribute addProperty Id "MTO_Inputs_Channel_1AT %I*MTO_Inputs_Channel_53C09E8B6MTO_Inputs_Channel_2AT %I*MTO_Inputs_Channel_53C09E8B6MTO_Inputs_Channel_3AT %I*MTO_Inputs_Channel_53C09E8B6MTO_Inputs_Channel_4AT %I*MTO_Inputs_Channel_53C09E8B6MTO_Inputs_Channel_5AT %I*MTO_Inputs_Channel_53C09E8B6MTO_Inputs_Channel_6AT %I*MTO_Inputs_Channel_53C09E8B6MTO_Inputs_Channel_7AT %I*MTO_Inputs_Channel_53C09E8B6MTO_Inputs_Channel_8AT %I*MTO_Inputs_Channel_53C09E8B6MTI_Inputs_10x_Channel_1AT %I*MTI_Inputs_10x_Channel_C3ED30FD56MTI_Inputs_10x_Channel_2AT %I*MTI_Inputs_10x_Channel_C3ED30FD56MTI_Inputs_10x_Channel_3AT %I*MTI_Inputs_10x_Channel_C3ED30FD56MTI_Inputs_10x_Channel_4AT %I*MTI_Inputs_10x_Channel_C3ED30FD56MTI_Inputs_10x_Channel_5AT %I*MTI_Inputs_10x_Channel_C3ED30FD56MTI_Inputs_10x_Channel_6AT %I*MTI_Inputs_10x_Channel_C3ED30FD56MTI_Inputs_10x_Channel_7AT %I*MTI_Inputs_10x_Channel_C3ED30FD56MTI_Inputs_10x_Channel_8AT %I*MTI_Inputs_10x_Channel_C3ED30FD56MTO_Outputs_10x_Channel_1AT %Q*MTO_Outputs_10x_Channel_A3C0C02256MTO_Outputs_10x_Channel_2AT %Q*MTO_Outputs_10x_Channel_A3C0C02256MTO_Outputs_10x_Channel_3AT %Q*MTO_Outputs_10x_Channel_A3C0C02256MTO_Outputs_10x_Channel_4AT %Q*MTO_Outputs_10x_Channel_A3C0C02256MTO_Outputs_10x_Channel_5AT %Q*MTO_Outputs_10x_Channel_A3C0C02256MTO_Outputs_10x_Channel_6AT %Q*MTO_Outputs_10x_Channel_A3C0C02256MTO_Outputs_10x_Channel_7AT %Q*MTO_Outputs_10x_Channel_A3C0C02256MTO_Outputs_10x_Channel_8AT %Q*MTO_Outputs_10x_Channel_A3C0C02256MTI_Outputs_Channel_1AT %Q*MTI_Outputs_Channel_0F1028A12MTI_Outputs_Channel_2AT %Q*MTI_Outputs_Channel_0F1028A12MTI_Outputs_Channel_3AT %Q*MTI_Outputs_Channel_0F1028A12MTI_Outputs_Channel_4AT %Q*MTI_Outputs_Channel_0F1028A12MTI_Outputs_Channel_5AT %Q*MTI_Outputs_Channel_0F1028A12MTI_Outputs_Channel_6AT %Q*MTI_Outputs_Channel_0F1028A12MTI_Outputs_Channel_7AT %Q*MTI_Outputs_Channel_0F1028A12MTI_Outputs_Channel_8AT %Q*MTI_Outputs_Channel_0F1028A12WcStateAT %I*WcState_9091E0EB2InfoDataAT %I*InfoData_BEF6B88E18"}
{attribute addProperty CRC "2870863100"}
{attribute addProperty Size "980"}
TYPE EL1259_AB1DE4FC EXTENDS EtcSlaveTerminalBase_947E5A46 :
STRUCT
	{attribute addProperty Name "MTO_Inputs_Channel_1"}
	MTO_Inputs_Channel_1 : MTO_Inputs_Channel_53C09E8B;
	{attribute addProperty Name "MTO_Inputs_Channel_2"}
	MTO_Inputs_Channel_2 : MTO_Inputs_Channel_53C09E8B;
	{attribute addProperty Name "MTO_Inputs_Channel_3"}
	MTO_Inputs_Channel_3 : MTO_Inputs_Channel_53C09E8B;
	{attribute addProperty Name "MTO_Inputs_Channel_4"}
	MTO_Inputs_Channel_4 : MTO_Inputs_Channel_53C09E8B;
	{attribute addProperty Name "MTO_Inputs_Channel_5"}
	MTO_Inputs_Channel_5 : MTO_Inputs_Channel_53C09E8B;
	{attribute addProperty Name "MTO_Inputs_Channel_6"}
	MTO_Inputs_Channel_6 : MTO_Inputs_Channel_53C09E8B;
	{attribute addProperty Name "MTO_Inputs_Channel_7"}
	MTO_Inputs_Channel_7 : MTO_Inputs_Channel_53C09E8B;
	{attribute addProperty Name "MTO_Inputs_Channel_8"}
	MTO_Inputs_Channel_8 : MTO_Inputs_Channel_53C09E8B;
	{attribute addProperty Name "MTI_Inputs_10x_Channel_1"}
	MTI_Inputs_10x_Channel_1 : MTI_Inputs_10x_Channel_C3ED30FD;
	{attribute addProperty Name "MTI_Inputs_10x_Channel_2"}
	MTI_Inputs_10x_Channel_2 : MTI_Inputs_10x_Channel_C3ED30FD;
	{attribute addProperty Name "MTI_Inputs_10x_Channel_3"}
	MTI_Inputs_10x_Channel_3 : MTI_Inputs_10x_Channel_C3ED30FD;
	{attribute addProperty Name "MTI_Inputs_10x_Channel_4"}
	MTI_Inputs_10x_Channel_4 : MTI_Inputs_10x_Channel_C3ED30FD;
	{attribute addProperty Name "MTI_Inputs_10x_Channel_5"}
	MTI_Inputs_10x_Channel_5 : MTI_Inputs_10x_Channel_C3ED30FD;
	{attribute addProperty Name "MTI_Inputs_10x_Channel_6"}
	MTI_Inputs_10x_Channel_6 : MTI_Inputs_10x_Channel_C3ED30FD;
	{attribute addProperty Name "MTI_Inputs_10x_Channel_7"}
	MTI_Inputs_10x_Channel_7 : MTI_Inputs_10x_Channel_C3ED30FD;
	{attribute addProperty Name "MTI_Inputs_10x_Channel_8"}
	MTI_Inputs_10x_Channel_8 : MTI_Inputs_10x_Channel_C3ED30FD;
	{attribute addProperty Name "MTO_Outputs_10x_Channel_1"}
	MTO_Outputs_10x_Channel_1 : MTO_Outputs_10x_Channel_A3C0C022;
	{attribute addProperty Name "MTO_Outputs_10x_Channel_2"}
	MTO_Outputs_10x_Channel_2 : MTO_Outputs_10x_Channel_A3C0C022;
	{attribute addProperty Name "MTO_Outputs_10x_Channel_3"}
	MTO_Outputs_10x_Channel_3 : MTO_Outputs_10x_Channel_A3C0C022;
	{attribute addProperty Name "MTO_Outputs_10x_Channel_4"}
	MTO_Outputs_10x_Channel_4 : MTO_Outputs_10x_Channel_A3C0C022;
	{attribute addProperty Name "MTO_Outputs_10x_Channel_5"}
	MTO_Outputs_10x_Channel_5 : MTO_Outputs_10x_Channel_A3C0C022;
	{attribute addProperty Name "MTO_Outputs_10x_Channel_6"}
	MTO_Outputs_10x_Channel_6 : MTO_Outputs_10x_Channel_A3C0C022;
	{attribute addProperty Name "MTO_Outputs_10x_Channel_7"}
	MTO_Outputs_10x_Channel_7 : MTO_Outputs_10x_Channel_A3C0C022;
	{attribute addProperty Name "MTO_Outputs_10x_Channel_8"}
	MTO_Outputs_10x_Channel_8 : MTO_Outputs_10x_Channel_A3C0C022;
	{attribute addProperty Name "MTI_Outputs_Channel_1"}
	MTI_Outputs_Channel_1 : MTI_Outputs_Channel_0F1028A1;
	{attribute addProperty Name "MTI_Outputs_Channel_2"}
	MTI_Outputs_Channel_2 : MTI_Outputs_Channel_0F1028A1;
	{attribute addProperty Name "MTI_Outputs_Channel_3"}
	MTI_Outputs_Channel_3 : MTI_Outputs_Channel_0F1028A1;
	{attribute addProperty Name "MTI_Outputs_Channel_4"}
	MTI_Outputs_Channel_4 : MTI_Outputs_Channel_0F1028A1;
	{attribute addProperty Name "MTI_Outputs_Channel_5"}
	MTI_Outputs_Channel_5 : MTI_Outputs_Channel_0F1028A1;
	{attribute addProperty Name "MTI_Outputs_Channel_6"}
	MTI_Outputs_Channel_6 : MTI_Outputs_Channel_0F1028A1;
	{attribute addProperty Name "MTI_Outputs_Channel_7"}
	MTI_Outputs_Channel_7 : MTI_Outputs_Channel_0F1028A1;
	{attribute addProperty Name "MTI_Outputs_Channel_8"}
	MTI_Outputs_Channel_8 : MTI_Outputs_Channel_0F1028A1;
	{attribute addProperty Name "WcState"}
	WcState : WcState_9091E0EB;
	{attribute addProperty Name "InfoData"}
	InfoData : InfoData_BEF6B88E;
END_STRUCT
END_TYPE

// ---- DUTs/IO/Boxes/EL1382_6CC2DB6A.TcDUT
{attribute 'GeneratedUsingTerminal: EL1382-0000-0016'}
{attribute addProperty BoxType "EL1382-0000-0016"}
{attribute addProperty Description "EL1382 2Ch. Dig. Input thermistor"}
{attribute addProperty Physics "KK"}
{attribute addProperty Id "Channel_1AT %I*Channel_31CEFA7F2Channel_2AT %I*Channel_31CEFA7F2WcStateAT %I*WcState_9091E0EB2InfoDataAT %I*InfoData_6F19DB2B2"}
{attribute addProperty CRC "1824709482"}
{attribute addProperty Size "8"}
TYPE EL1382_6CC2DB6A EXTENDS EtcSlaveTerminalBase_947E5A46 :
STRUCT
	{attribute addProperty Name "Channel_1"}
	Channel_1 : Channel_31CEFA7F;
	{attribute addProperty Name "Channel_2"}
	Channel_2 : Channel_31CEFA7F;
	{attribute addProperty Name "WcState"}
	WcState : WcState_9091E0EB;
	{attribute addProperty Name "InfoData"}
	InfoData : InfoData_6F19DB2B;
END_STRUCT
END_TYPE

// ---- DUTs/IO/Boxes/EL1702_02444DCB.TcDUT
{attribute 'GeneratedUsingTerminal: EL1702-0000-0016'}
{attribute addProperty BoxType "EL1702-0000-0016"}
{attribute addProperty Description "EL1702 2Ch. Dig. Input 120V/230V AC, 10ms"}
{attribute addProperty Physics "KK"}
{attribute addProperty Id "Channel_1AT %I*Channel_830843C11Channel_2AT %I*Channel_830843C11WcStateAT %I*WcState_9091E0EB2InfoDataAT %I*InfoData_6F19DB2B2"}
{attribute addProperty CRC "38030795"}
{attribute addProperty Size "6"}
TYPE EL1702_02444DCB EXTENDS EtcSlaveTerminalBase_947E5A46 :
STRUCT
	{attribute addProperty Name "Channel_1"}
	Channel_1 : Channel_830843C1;
	{attribute addProperty Name "Channel_2"}
	Channel_2 : Channel_830843C1;
	{attribute addProperty Name "WcState"}
	WcState : WcState_9091E0EB;
	{attribute addProperty Name "InfoData"}
	InfoData : InfoData_6F19DB2B;
END_STRUCT
END_TYPE

// ---- DUTs/IO/Boxes/EL1712_02444DCB.TcDUT
{attribute 'GeneratedUsingTerminal: EL1712-0000-0016'}
{attribute addProperty BoxType "EL1712-0000-0016"}
{attribute addProperty Description "EL1712 2Ch. Dig. Input 120V AC/DC, 10ms"}
{attribute addProperty Physics "KK"}
{attribute addProperty Id "Channel_1AT %I*Channel_830843C11Channel_2AT %I*Channel_830843C11WcStateAT %I*WcState_9091E0EB2InfoDataAT %I*InfoData_6F19DB2B2"}
{attribute addProperty CRC "38030795"}
{attribute addProperty Size "6"}
TYPE EL1712_02444DCB EXTENDS EtcSlaveTerminalBase_947E5A46 :
STRUCT
	{attribute addProperty Name "Channel_1"}
	Channel_1 : Channel_830843C1;
	{attribute addProperty Name "Channel_2"}
	Channel_2 : Channel_830843C1;
	{attribute addProperty Name "WcState"}
	WcState : WcState_9091E0EB;
	{attribute addProperty Name "InfoData"}
	InfoData : InfoData_6F19DB2B;
END_STRUCT
END_TYPE

// ---- DUTs/IO/Boxes/EL1722_02444DCB.TcDUT
{attribute 'GeneratedUsingTerminal: EL1722-0000-0016'}
{attribute addProperty BoxType "EL1722-0000-0016"}
{attribute addProperty Description "EL1722 2Ch. Dig. Input 120V/230V AC, 10ms, no power contacts"}
{attribute addProperty Physics "KK"}
{attribute addProperty Id "Channel_1AT %I*Channel_830843C11Channel_2AT %I*Channel_830843C11WcStateAT %I*WcState_9091E0EB2InfoDataAT %I*InfoData_6F19DB2B2"}
{attribute addProperty CRC "38030795"}
{attribute addProperty Size "6"}
TYPE EL1722_02444DCB EXTENDS EtcSlaveTerminalBase_947E5A46 :
STRUCT
	{attribute addProperty Name "Channel_1"}
	Channel_1 : Channel_830843C1;
	{attribute addProperty Name "Channel_2"}
	Channel_2 : Channel_830843C1;
	{attribute addProperty Name "WcState"}
	WcState : WcState_9091E0EB;
	{attribute addProperty Name "InfoData"}
	InfoData : InfoData_6F19DB2B;
END_STRUCT
END_TYPE

// ---- DUTs/IO/Boxes/EL1804_D135F8DB.TcDUT
{attribute 'GeneratedUsingTerminal: EL1804-0000-0016'}
{attribute addProperty BoxType "EL1804-0000-0016"}
{attribute addProperty Description "EL1804 4Ch. Dig. Input 24V, 3ms"}
{attribute addProperty Physics "KK"}
{attribute addProperty Id "Channel_1AT %I*Channel_830843C11Channel_2AT %I*Channel_830843C11Channel_3AT %I*Channel_830843C11Channel_4AT %I*Channel_830843C11WcStateAT %I*WcState_9091E0EB2InfoDataAT %I*InfoData_6F19DB2B2"}
{attribute addProperty CRC "3509975259"}
{attribute addProperty Size "8"}
TYPE EL1804_D135F8DB EXTENDS EtcSlaveTerminalBase_947E5A46 :
STRUCT
	{attribute addProperty Name "Channel_1"}
	Channel_1 : Channel_830843C1;
	{attribute addProperty Name "Channel_2"}
	Channel_2 : Channel_830843C1;
	{attribute addProperty Name "Channel_3"}
	Channel_3 : Channel_830843C1;
	{attribute addProperty Name "Channel_4"}
	Channel_4 : Channel_830843C1;
	{attribute addProperty Name "WcState"}
	WcState : WcState_9091E0EB;
	{attribute addProperty Name "InfoData"}
	InfoData : InfoData_6F19DB2B;
END_STRUCT
END_TYPE

